LIN {X 0,Y 574.928,Z 413.278,A -85,B 0,C 180,E1 -2269.45,E2 -2269.45} C_VEL
LIN {X 0,Y 575.117,Z 397.956,A -85,B 0,C 180,E1 -2270.055,E2 -2270.055} C_VEL
LIN {X 0,Y 575.352,Z 381.203,A -85,B 0,C 180,E1 -2270.559,E2 -2270.559} C_VEL
LIN {X 0,Y 575.53,Z 364.973,A -85,B 0,C 180,E1 -2270.903,E2 -2270.903} C_VEL
LIN {X 0,Y 576.146,Z 164.419,A -85,B 0,C 180,E1 -2273.543,E2 -2273.543} C_VEL
LIN {X 0,Y 575.13,Z 158.184,A -85,B 0,C 180,E1 -2273.687,E2 -2273.687} C_VEL
LIN {X 0,Y 575.609,Z 123.808,A -85,B 0,C 180,E1 -2276.367,E2 -2276.367} C_VEL
LIN {X 0,Y 575.922,Z 94.132,A -85,B 0,C 180,E1 -2278.717,E2 -2278.717} C_VEL
LIN {X 0,Y 573.276,Z 85.388,A -85,B 0,C 180,E1 -2279.565,E2 -2279.565} C_VEL
LIN {X 0,Y 573.253,Z 85.395,A -85,B 0,C 180,E1 -2282.644,E2 -2282.644} C_VEL
LIN {X 0,Y 573.208,Z 85.394,A -85,B 0,C 180,E1 -2285.187,E2 -2285.187} C_VEL
LIN {X 0,Y 573.23,Z 85.39,A -85,B 0,C 180,E1 -2287.807,E2 -2287.807} C_VEL
LIN {X 0,Y 573.24,Z 85.397,A -85,B 0,C 180,E1 -2290.525,E2 -2290.525} C_VEL
LIN {X 0,Y 573.244,Z 85.387,A -85,B 0,C 180,E1 -2293.358,E2 -2293.358} C_VEL
LIN {X 0,Y 573.24,Z 85.396,A -85,B 0,C 180,E1 -2296.331,E2 -2296.331} C_VEL
LIN {X 0,Y 573.27,Z 85.383,A -85,B 0,C 180,E1 -2299.477,E2 -2299.477} C_VEL
LIN {X 0,Y 573.232,Z 85.396,A -85,B 0,C 180,E1 -2302.192,E2 -2302.192} C_VEL
LIN {X 0,Y 573.263,Z 85.385,A -85,B 0,C 180,E1 -2304.816,E2 -2304.816} C_VEL
LIN {X 0,Y 573.25,Z 85.385,A -85,B 0,C 180,E1 -2307.355,E2 -2307.355} C_VEL
LIN {X 0,Y 573.246,Z 85.39,A -85,B 0,C 180,E1 -2309.824,E2 -2309.824} C_VEL
LIN {X 0,Y 573.269,Z 85.391,A -85,B 0,C 180,E1 -2312.234,E2 -2312.234} C_VEL
LIN {X 0,Y 573.264,Z 85.383,A -85,B 0,C 180,E1 -2315.121,E2 -2315.121} C_VEL
LIN {X 0,Y 573.233,Z 85.392,A -85,B 0,C 180,E1 -2317.662,E2 -2317.662} C_VEL
LIN {X 0,Y 573.274,Z 85.383,A -85,B 0,C 180,E1 -2320.728,E2 -2320.728} C_VEL
LIN {X 0,Y 573.248,Z 85.391,A -85,B 0,C 180,E1 -2323.622,E2 -2323.622} C_VEL
LIN {X 0,Y 573.27,Z 85.392,A -85,B 0,C 180,E1 -2325.807,E2 -2325.807} C_VEL
LIN {X 0,Y 573.258,Z 85.384,A -85,B 0,C 180,E1 -2328.745,E2 -2328.745} C_VEL
LIN {X 0,Y 573.281,Z 85.387,A -85,B 0,C 180,E1 -2331.541,E2 -2331.541} C_VEL
LIN {X 0,Y 573.287,Z 85.382,A -85,B 0,C 180,E1 -2334.372,E2 -2334.372} C_VEL
LIN {X 0,Y 573.305,Z 85.385,A -85,B 0,C 180,E1 -2337.892,E2 -2337.892} C_VEL
LIN {X 0,Y 573.329,Z 85.375,A -85,B 0,C 180,E1 -2340.702,E2 -2340.702} C_VEL
LIN {X 0,Y 573.232,Z 85.397,A -85,B 0,C 180,E1 -2343.515,E2 -2343.515} C_VEL
LIN {X 0,Y 573.285,Z 85.389,A -85,B 0,C 180,E1 -2345.628,E2 -2345.628} C_VEL
LIN {X 0,Y 573.28,Z 85.381,A -85,B 0,C 180,E1 -2348.46,E2 -2348.46} C_VEL
LIN {X 0,Y 573.268,Z 85.391,A -85,B 0,C 180,E1 -2351.312,E2 -2351.312} C_VEL
LIN {X 0,Y 573.269,Z 85.383,A -85,B 0,C 180,E1 -2354.193,E2 -2354.193} C_VEL
LIN {X 0,Y 573.256,Z 85.391,A -85,B 0,C 180,E1 -2357.112,E2 -2357.112} C_VEL
LIN {X 0,Y 573.248,Z 85.386,A -85,B 0,C 180,E1 -2360.077,E2 -2360.077} C_VEL
LIN {X 0,Y 573.23,Z 85.396,A -85,B 0,C 180,E1 -2363.1,E2 -2363.1} C_VEL
LIN {X 0,Y 573.247,Z 85.386,A -85,B 0,C 180,E1 -2364.39,E2 -2364.39} C_VEL
LIN {X 0,Y 572.62,Z 85.471,A -85,B 0,C 180,E1 -2364.977,E2 -2364.977} C_VEL
LIN {X 0,Y 569.778,Z 85.828,A -85,B 0,C 180,E1 -2365.928,E2 -2365.928} C_VEL
LIN {X 0,Y 567.346,Z 86.132,A -85,B 0,C 180,E1 -2366.694,E2 -2366.694} C_VEL
LIN {X 0,Y 566.29,Z 86.26,A -85,B 0,C 180,E1 -2367.285,E2 -2367.285} C_VEL
LIN {X 0,Y 566.2,Z 86.268,A -85,B 0,C 180,E1 -2367.485,E2 -2367.485} C_VEL
LIN {X 0,Y 566.198,Z 86.265,A -85,B 0,C 180,E1 -2369.769,E2 -2369.769} C_VEL
LIN {X 0,Y 566.202,Z 86.265,A -85,B 0,C 180,E1 -2372.431,E2 -2372.431} C_VEL
LIN {X 0,Y 566.209,Z 86.272,A -85,B 0,C 180,E1 -2374.995,E2 -2374.995} C_VEL
LIN {X 0,Y 566.194,Z 86.267,A -85,B 0,C 180,E1 -2377.461,E2 -2377.461} C_VEL
LIN {X 0,Y 566.224,Z 86.261,A -85,B 0,C 180,E1 -2380.198,E2 -2380.198} C_VEL
LIN {X 0,Y 566.198,Z 86.271,A -85,B 0,C 180,E1 -2383.054,E2 -2383.054} C_VEL
LIN {X 0,Y 566.199,Z 86.264,A -85,B 0,C 180,E1 -2386.049,E2 -2386.049} C_VEL
LIN {X 0,Y 566.209,Z 86.271,A -85,B 0,C 180,E1 -2388.864,E2 -2388.864} C_VEL
LIN {X 0,Y 566.186,Z 86.265,A -85,B 0,C 180,E1 -2391.638,E2 -2391.638} C_VEL
LIN {X 0,Y 566.16,Z 86.272,A -85,B 0,C 180,E1 -2394.308,E2 -2394.308} C_VEL
LIN {X 0,Y 566.228,Z 86.266,A -85,B 0,C 180,E1 -2396.899,E2 -2396.899} C_VEL
LIN {X 0,Y 566.183,Z 86.266,A -85,B 0,C 180,E1 -2399.408,E2 -2399.408} C_VEL
LIN {X 0,Y 566.21,Z 86.263,A -85,B 0,C 180,E1 -2401.858,E2 -2401.858} C_VEL
LIN {X 0,Y 566.213,Z 86.268,A -85,B 0,C 180,E1 -2404.252,E2 -2404.252} C_VEL
LIN {X 0,Y 566.171,Z 86.273,A -85,B 0,C 180,E1 -2406.719,E2 -2406.719} C_VEL
LIN {X 0,Y 566.212,Z 86.263,A -85,B 0,C 180,E1 -2409.663,E2 -2409.663} C_VEL
LIN {X 0,Y 566.199,Z 86.269,A -85,B 0,C 180,E1 -2412.669,E2 -2412.669} C_VEL
LIN {X 0,Y 566.234,Z 86.26,A -85,B 0,C 180,E1 -2415.627,E2 -2415.627} C_VEL
LIN {X 0,Y 566.235,Z 86.263,A -85,B 0,C 180,E1 -2418.676,E2 -2418.676} C_VEL
LIN {X 0,Y 566.227,Z 86.261,A -85,B 0,C 180,E1 -2421.435,E2 -2421.435} C_VEL
LIN {X 0,Y 566.259,Z 86.264,A -85,B 0,C 180,E1 -2424.302,E2 -2424.302} C_VEL
LIN {X 0,Y 566.283,Z 86.259,A -85,B 0,C 180,E1 -2427.867,E2 -2427.867} C_VEL
LIN {X 0,Y 566.302,Z 86.252,A -85,B 0,C 180,E1 -2430.712,E2 -2430.712} C_VEL
LIN {X 0,Y 566.271,Z 86.255,A -85,B 0,C 180,E1 -2432.846,E2 -2432.846} C_VEL
LIN {X 0,Y 566.258,Z 86.262,A -85,B 0,C 180,E1 -2435.699,E2 -2435.699} C_VEL
LIN {X 0,Y 566.229,Z 86.261,A -85,B 0,C 180,E1 -2438.566,E2 -2438.566} C_VEL
LIN {X 0,Y 566.244,Z 86.262,A -85,B 0,C 180,E1 -2441.455,E2 -2441.455} C_VEL
LIN {X 0,Y 566.236,Z 86.26,A -85,B 0,C 180,E1 -2444.507,E2 -2444.507} C_VEL
LIN {X 0,Y 566.201,Z 86.267,A -85,B 0,C 180,E1 -2447.332,E2 -2447.332} C_VEL
LIN {X 0,Y 566.214,Z 86.263,A -85,B 0,C 180,E1 -2450.338,E2 -2450.338} C_VEL
LIN {X 0,Y 566.175,Z 86.271,A -85,B 0,C 180,E1 -2453.282,E2 -2453.282} C_VEL
LIN {X 0,Y 566.217,Z 86.269,A -85,B 0,C 180,E1 -2455.749,E2 -2455.749} C_VEL
LIN {X 0,Y 566.205,Z 86.264,A -85,B 0,C 180,E1 -2458.202,E2 -2458.202} C_VEL
LIN {X 0,Y 566.192,Z 86.268,A -85,B 0,C 180,E1 -2461.077,E2 -2461.077} C_VEL
LIN {X 0,Y 566.214,Z 86.267,A -85,B 0,C 180,E1 -2463.734,E2 -2463.734} C_VEL
LIN {X 0,Y 566.201,Z 86.264,A -85,B 0,C 180,E1 -2466.57,E2 -2466.57} C_VEL
LIN {X 0,Y 566.216,Z 86.266,A -85,B 0,C 180,E1 -2469.686,E2 -2469.686} C_VEL
LIN {X 0,Y 566.205,Z 86.267,A -85,B 0,C 180,E1 -2472.918,E2 -2472.918} C_VEL
LIN {X 0,Y 566.197,Z 86.264,A -85,B 0,C 180,E1 -2476.049,E2 -2476.049} C_VEL
LIN {X 0,Y 566.206,Z 86.273,A -85,B 0,C 180,E1 -2479.215,E2 -2479.215} C_VEL
LIN {X 0,Y 566.189,Z 86.268,A -85,B 0,C 180,E1 -2481.637,E2 -2481.637} C_VEL
LIN {X 0,Y 566.195,Z 86.265,A -85,B 0,C 180,E1 -2484.31,E2 -2484.31} C_VEL
LIN {X 0,Y 566.223,Z 86.268,A -85,B 0,C 180,E1 -2486.898,E2 -2486.898} C_VEL
LIN {X 0,Y 566.184,Z 86.271,A -85,B 0,C 180,E1 -2489.407,E2 -2489.407} C_VEL
LIN {X 0,Y 566.216,Z 86.264,A -85,B 0,C 180,E1 -2491.858,E2 -2491.858} C_VEL
LIN {X 0,Y 566.213,Z 86.266,A -85,B 0,C 180,E1 -2494.251,E2 -2494.251} C_VEL
LIN {X 0,Y 566.197,Z 86.269,A -85,B 0,C 180,E1 -2496.075,E2 -2496.075} C_VEL
LIN {X 0,Y 567.227,Z 89.177,A -85,B 0,C 180,E1 -2496.169,E2 -2496.169} C_VEL
LIN {X 0,Y 569.661,Z 94.835,A -85,B 0,C 180,E1 -2496.361,E2 -2496.361} C_VEL
LIN {X 0,Y 568.867,Z 283.383,A -85,B 0,C 180,E1 -2498.863,E2 -2498.863} C_VEL
LIN {X 0,Y 568.754,Z 299.599,A -85,B 0,C 180,E1 -2499.191,E2 -2499.191} C_VEL
LIN {X 0,Y 568.499,Z 315.266,A -85,B 0,C 180,E1 -2499.654,E2 -2499.654} C_VEL
LIN {X 0,Y 568.295,Z 327.963,A -85,B 0,C 180,E1 -2500.132,E2 -2500.132} C_VEL
LIN {X 0,Y 567.998,Z 341.858,A -85,B 0,C 180,E1 -2500.765,E2 -2500.765} C_VEL
LIN {X 0,Y 567.689,Z 356.768,A -85,B 0,C 180,E1 -2501.597,E2 -2501.597} C_VEL
LIN {X 0,Y 567.395,Z 369.444,A -85,B 0,C 180,E1 -2502.444,E2 -2502.444} C_VEL
LIN {X 0,Y 567.154,Z 381.162,A -85,B 0,C 180,E1 -2503.348,E2 -2503.348} C_VEL
LIN {X 0,Y 566.863,Z 392.522,A -85,B 0,C 180,E1 -2504.356,E2 -2504.356} C_VEL
LIN {X 0,Y 566.634,Z 404.905,A -85,B 0,C 180,E1 -2505.637,E2 -2505.637} C_VEL
LIN {X 0,Y 566.379,Z 415.329,A -85,B 0,C 180,E1 -2506.911,E2 -2506.911} C_VEL
LIN {X 0,Y 566.221,Z 424.31,A -85,B 0,C 180,E1 -2508.182,E2 -2508.182} C_VEL
LIN {X 0,Y 566.118,Z 432.007,A -85,B 0,C 180,E1 -2509.449,E2 -2509.449} C_VEL
LIN {X 0,Y 566.005,Z 438.589,A -85,B 0,C 180,E1 -2510.711,E2 -2510.711} C_VEL
LIN {X 0,Y 565.979,Z 444.894,A -85,B 0,C 180,E1 -2512.149,E2 -2512.149} C_VEL
LIN {X 0,Y 565.92,Z 449.999,A -85,B 0,C 180,E1 -2513.583,E2 -2513.583} C_VEL
LIN {X 0,Y 565.86,Z 453.972,A -85,B 0,C 180,E1 -2515.012,E2 -2515.012} C_VEL
LIN {X 0,Y 565.911,Z 456.887,A -85,B 0,C 180,E1 -2516.44,E2 -2516.44} C_VEL
LIN {X 0,Y 565.829,Z 458.84,A -85,B 0,C 180,E1 -2517.864,E2 -2517.864} C_VEL
LIN {X 0,Y 565.839,Z 459.811,A -85,B 0,C 180,E1 -2519.288,E2 -2519.288} C_VEL
LIN {X 0,Y 565.841,Z 459.839,A -85,B 0,C 180,E1 -2520.712,E2 -2520.712} C_VEL
LIN {X 0,Y 565.829,Z 458.925,A -85,B 0,C 180,E1 -2522.135,E2 -2522.135} C_VEL
LIN {X 0,Y 565.91,Z 457.029,A -85,B 0,C 180,E1 -2523.56,E2 -2523.56} C_VEL
LIN {X 0,Y 565.858,Z 454.187,A -85,B 0,C 180,E1 -2524.988,E2 -2524.988} C_VEL
LIN {X 0,Y 565.948,Z 449.836,A -85,B 0,C 180,E1 -2526.56,E2 -2526.56} C_VEL
LIN {X 0,Y 565.99,Z 443.787,A -85,B 0,C 180,E1 -2528.21,E2 -2528.21} C_VEL
LIN {X 0,Y 566.034,Z 437.256,A -85,B 0,C 180,E1 -2529.649,E2 -2529.649} C_VEL
LIN {X 0,Y 566.18,Z 429.121,A -85,B 0,C 180,E1 -2531.147,E2 -2531.147} C_VEL
LIN {X 0,Y 566.322,Z 420.049,A -85,B 0,C 180,E1 -2532.543,E2 -2532.543} C_VEL
LIN {X 0,Y 566.514,Z 410.291,A -85,B 0,C 180,E1 -2533.816,E2 -2533.816} C_VEL
LIN {X 0,Y 566.701,Z 400.453,A -85,B 0,C 180,E1 -2534.932,E2 -2534.932} C_VEL
LIN {X 0,Y 566.901,Z 391.505,A -85,B 0,C 180,E1 -2535.827,E2 -2535.827} C_VEL
LIN {X 0,Y 567.147,Z 380.013,A -85,B 0,C 180,E1 -2536.837,E2 -2536.837} C_VEL
LIN {X 0,Y 567.449,Z 367.853,A -85,B 0,C 180,E1 -2537.761,E2 -2537.761} C_VEL
LIN {X 0,Y 567.762,Z 353.698,A -85,B 0,C 180,E1 -2538.68,E2 -2538.68} C_VEL
LIN {X 0,Y 568.039,Z 339.87,A -85,B 0,C 180,E1 -2539.421,E2 -2539.421} C_VEL
LIN {X 0,Y 568.304,Z 326.571,A -85,B 0,C 180,E1 -2540.017,E2 -2540.017} C_VEL
LIN {X 0,Y 568.611,Z 310.214,A -85,B 0,C 180,E1 -2540.602,E2 -2540.602} C_VEL
LIN {X 0,Y 568.775,Z 295.187,A -85,B 0,C 180,E1 -2540.998,E2 -2540.998} C_VEL
LIN {X 0,Y 568.884,Z 281.636,A -85,B 0,C 180,E1 -2541.254,E2 -2541.254} C_VEL
LIN {X 0,Y 569.594,Z 95.156,A -85,B 0,C 180,E1 -2543.726,E2 -2543.726} C_VEL
LIN {X 0,Y 569.036,Z 93.275,A -85,B 0,C 180,E1 -2543.778,E2 -2543.778} C_VEL
LIN {X 0,Y 566.316,Z 87.098,A -85,B 0,C 180,E1 -2543.991,E2 -2543.991} C_VEL
LIN {X 0,Y 566.14,Z 86.277,A -85,B 0,C 180,E1 -2544.028,E2 -2544.028} C_VEL
LIN {X 0,Y 566.169,Z 86.275,A -85,B 0,C 180,E1 -2546.65,E2 -2546.65} C_VEL
LIN {X 0,Y 566.158,Z 86.272,A -85,B 0,C 180,E1 -2549.771,E2 -2549.771} C_VEL
LIN {X 0,Y 566.194,Z 86.272,A -85,B 0,C 180,E1 -2552.428,E2 -2552.428} C_VEL
LIN {X 0,Y 566.178,Z 86.272,A -85,B 0,C 180,E1 -2554.989,E2 -2554.989} C_VEL
LIN {X 0,Y 566.192,Z 86.267,A -85,B 0,C 180,E1 -2557.461,E2 -2557.461} C_VEL
LIN {X 0,Y 566.207,Z 86.271,A -85,B 0,C 180,E1 -2560.199,E2 -2560.199} C_VEL
LIN {X 0,Y 566.198,Z 86.266,A -85,B 0,C 180,E1 -2563.054,E2 -2563.054} C_VEL
LIN {X 0,Y 566.2,Z 86.273,A -85,B 0,C 180,E1 -2566.048,E2 -2566.048} C_VEL
LIN {X 0,Y 566.205,Z 86.266,A -85,B 0,C 180,E1 -2569.214,E2 -2569.214} C_VEL
LIN {X 0,Y 566.188,Z 86.274,A -85,B 0,C 180,E1 -2571.636,E2 -2571.636} C_VEL
LIN {X 0,Y 566.164,Z 86.273,A -85,B 0,C 180,E1 -2574.308,E2 -2574.308} C_VEL
LIN {X 0,Y 566.23,Z 86.267,A -85,B 0,C 180,E1 -2576.898,E2 -2576.898} C_VEL
LIN {X 0,Y 566.182,Z 86.279,A -85,B 0,C 180,E1 -2579.407,E2 -2579.407} C_VEL
LIN {X 0,Y 566.226,Z 86.394,A -85,B 0,C 180,E1 -2580.324,E2 -2580.324} C_VEL
LIN {X 0,Y 569.015,Z 96.641,A -85,B 0,C 180,E1 -2581.274,E2 -2581.274} C_VEL
LIN {X 0,Y 568.654,Z 132.486,A -85,B 0,C 180,E1 -2584.074,E2 -2584.074} C_VEL
LIN {X 0,Y 568.402,Z 157.927,A -85,B 0,C 180,E1 -2586.031,E2 -2586.031} C_VEL
LIN {X 0,Y 569.69,Z 167.303,A -85,B 0,C 180,E1 -2586.217,E2 -2586.217} C_VEL
LIN {X 0,Y 568.884,Z 364.907,A -85,B 0,C 180,E1 -2588.84,E2 -2588.84} C_VEL
LIN {X 0,Y 568.702,Z 381.158,A -85,B 0,C 180,E1 -2589.188,E2 -2589.188} C_VEL
LIN {X 0,Y 568.44,Z 397.926,A -85,B 0,C 180,E1 -2589.698,E2 -2589.698} C_VEL
LIN {X 0,Y 568.206,Z 413.659,A -85,B 0,C 180,E1 -2590.329,E2 -2590.329} C_VEL
LIN {X 0,Y 567.901,Z 428.026,A -85,B 0,C 180,E1 -2591.043,E2 -2591.043} C_VEL
LIN {X 0,Y 567.532,Z 443.265,A -85,B 0,C 180,E1 -2591.965,E2 -2591.965} C_VEL
LIN {X 0,Y 567.19,Z 457.209,A -85,B 0,C 180,E1 -2592.978,E2 -2592.978} C_VEL
LIN {X 0,Y 566.916,Z 471.063,A -85,B 0,C 180,E1 -2594.173,E2 -2594.173} C_VEL
LIN {X 0,Y 566.632,Z 482.615,A -85,B 0,C 180,E1 -2595.339,E2 -2595.339} C_VEL
LIN {X 0,Y 566.435,Z 494.334,A -85,B 0,C 180,E1 -2596.73,E2 -2596.73} C_VEL
LIN {X 0,Y 566.239,Z 504.668,A -85,B 0,C 180,E1 -2598.182,E2 -2598.182} C_VEL
LIN {X 0,Y 566.124,Z 513.281,A -85,B 0,C 180,E1 -2599.629,E2 -2599.629} C_VEL
LIN {X 0,Y 566.002,Z 520.488,A -85,B 0,C 180,E1 -2601.07,E2 -2601.07} C_VEL
LIN {X 0,Y 565.967,Z 526.464,A -85,B 0,C 180,E1 -2602.508,E2 -2602.508} C_VEL
LIN {X 0,Y 565.916,Z 531.186,A -85,B 0,C 180,E1 -2603.94,E2 -2603.94} C_VEL
LIN {X 0,Y 565.91,Z 535.635,A -85,B 0,C 180,E1 -2605.726,E2 -2605.726} C_VEL
LIN {X 0,Y 565.867,Z 538.089,A -85,B 0,C 180,E1 -2607.152,E2 -2607.152} C_VEL
LIN {X 0,Y 565.843,Z 539.479,A -85,B 0,C 180,E1 -2608.576,E2 -2608.576} C_VEL
LIN {X 0,Y 565.834,Z 540,A -85,B 0,C 180,E1 -2610,E2 -2610} C_VEL
LIN {X 0,Y 565.843,Z 539.48,A -85,B 0,C 180,E1 -2611.423,E2 -2611.423} C_VEL
LIN {X 0,Y 565.867,Z 538.089,A -85,B 0,C 180,E1 -2612.847,E2 -2612.847} C_VEL
LIN {X 0,Y 565.91,Z 535.637,A -85,B 0,C 180,E1 -2614.273,E2 -2614.273} C_VEL
LIN {X 0,Y 565.915,Z 531.19,A -85,B 0,C 180,E1 -2616.059,E2 -2616.059} C_VEL
LIN {X 0,Y 565.969,Z 526.47,A -85,B 0,C 180,E1 -2617.491,E2 -2617.491} C_VEL
LIN {X 0,Y 566.011,Z 520.492,A -85,B 0,C 180,E1 -2618.928,E2 -2618.928} C_VEL
LIN {X 0,Y 566.123,Z 513.286,A -85,B 0,C 180,E1 -2620.37,E2 -2620.37} C_VEL
LIN {X 0,Y 566.237,Z 504.676,A -85,B 0,C 180,E1 -2621.817,E2 -2621.817} C_VEL
LIN {X 0,Y 566.434,Z 494.342,A -85,B 0,C 180,E1 -2623.269,E2 -2623.269} C_VEL
LIN {X 0,Y 566.617,Z 482.669,A -85,B 0,C 180,E1 -2624.655,E2 -2624.655} C_VEL
LIN {X 0,Y 566.914,Z 471.072,A -85,B 0,C 180,E1 -2625.826,E2 -2625.826} C_VEL
LIN {X 0,Y 567.223,Z 457.222,A -85,B 0,C 180,E1 -2627.02,E2 -2627.02} C_VEL
LIN {X 0,Y 567.581,Z 443.28,A -85,B 0,C 180,E1 -2628.032,E2 -2628.032} C_VEL
LIN {X 0,Y 567.877,Z 429.716,A -85,B 0,C 180,E1 -2628.863,E2 -2628.863} C_VEL
LIN {X 0,Y 568.154,Z 415.368,A -85,B 0,C 180,E1 -2629.592,E2 -2629.592} C_VEL
LIN {X 0,Y 568.42,Z 399.254,A -85,B 0,C 180,E1 -2630.254,E2 -2630.254} C_VEL
LIN {X 0,Y 568.726,Z 383.034,A -85,B 0,C 180,E1 -2630.762,E2 -2630.762} C_VEL
LIN {X 0,Y 568.892,Z 366.461,A -85,B 0,C 180,E1 -2631.135,E2 -2631.135} C_VEL
LIN {X 0,Y 569.65,Z 175.195,A -85,B 0,C 180,E1 -2633.678,E2 -2633.678} C_VEL
LIN {X 0,Y 569.486,Z 164.584,A -85,B 0,C 180,E1 -2633.827,E2 -2633.827} C_VEL
LIN {X 0,Y 568.424,Z 158.163,A -85,B 0,C 180,E1 -2633.969,E2 -2633.969} C_VEL
LIN {X 0,Y 568.936,Z 123.563,A -85,B 0,C 180,E1 -2636.689,E2 -2636.689} C_VEL
LIN {X 0,Y 569.296,Z 96.342,A -85,B 0,C 180,E1 -2638.871,E2 -2638.871} C_VEL
LIN {X 0,Y 566.225,Z 86.267,A -85,B 0,C 180,E1 -2639.869,E2 -2639.869} C_VEL
LIN {X 0,Y 566.226,Z 86.266,A -85,B 0,C 180,E1 -2643.101,E2 -2643.101} C_VEL
LIN {X 0,Y 566.161,Z 86.27,A -85,B 0,C 180,E1 -2645.692,E2 -2645.692} C_VEL
LIN {X 0,Y 566.207,Z 86.273,A -85,B 0,C 180,E1 -2648.558,E2 -2648.558} C_VEL
LIN {X 0,Y 566.179,Z 86.268,A -85,B 0,C 180,E1 -2651.138,E2 -2651.138} C_VEL
LIN {X 0,Y 566.196,Z 86.268,A -85,B 0,C 180,E1 -2654.035,E2 -2654.035} C_VEL
LIN {X 0,Y 566.197,Z 86.265,A -85,B 0,C 180,E1 -2657.083,E2 -2657.083} C_VEL
LIN {X 0,Y 566.223,Z 86.263,A -85,B 0,C 180,E1 -2659.802,E2 -2659.802} C_VEL
LIN {X 0,Y 566.194,Z 86.269,A -85,B 0,C 180,E1 -2662.599,E2 -2662.599} C_VEL
LIN {X 0,Y 566.216,Z 86.261,A -85,B 0,C 180,E1 -2665.183,E2 -2665.183} C_VEL
LIN {X 0,Y 566.228,Z 86.263,A -85,B 0,C 180,E1 -2667.743,E2 -2667.743} C_VEL
LIN {X 0,Y 566.2,Z 86.27,A -85,B 0,C 180,E1 -2670.328,E2 -2670.328} C_VEL
LIN {X 0,Y 566.207,Z 86.263,A -85,B 0,C 180,E1 -2673.34,E2 -2673.34} C_VEL
LIN {X 0,Y 566.195,Z 86.27,A -85,B 0,C 180,E1 -2675.819,E2 -2675.819} C_VEL
LIN {X 0,Y 566.204,Z 86.263,A -85,B 0,C 180,E1 -2678.902,E2 -2678.902} C_VEL
LIN {X 0,Y 566.204,Z 86.263,A -85,B 0,C 180,E1 -2681.172,E2 -2681.172} C_VEL
LIN {X 0,Y 566.212,Z 86.264,A -85,B 0,C 180,E1 -2683.412,E2 -2683.412} C_VEL
LIN {X 0,Y 566.196,Z 86.267,A -85,B 0,C 180,E1 -2686.359,E2 -2686.359} C_VEL
LIN {X 0,Y 566.23,Z 86.26,A -85,B 0,C 180,E1 -2688.675,E2 -2688.675} C_VEL
LIN {X 0,Y 566.224,Z 86.265,A -85,B 0,C 180,E1 -2691.434,E2 -2691.434} C_VEL
LIN {X 0,Y 566.255,Z 86.258,A -85,B 0,C 180,E1 -2694.302,E2 -2694.302} C_VEL
LIN {X 0,Y 566.276,Z 86.261,A -85,B 0,C 180,E1 -2697.866,E2 -2697.866} C_VEL
LIN {X 0,Y 566.299,Z 86.251,A -85,B 0,C 180,E1 -2700.711,E2 -2700.711} C_VEL
LIN {X 0,Y 566.27,Z 86.255,A -85,B 0,C 180,E1 -2702.846,E2 -2702.846} C_VEL
LIN {X 0,Y 566.253,Z 86.264,A -85,B 0,C 180,E1 -2705.698,E2 -2705.698} C_VEL
LIN {X 0,Y 566.224,Z 86.261,A -85,B 0,C 180,E1 -2708.566,E2 -2708.566} C_VEL
LIN {X 0,Y 566.238,Z 86.269,A -85,B 0,C 180,E1 -2711.454,E2 -2711.454} C_VEL
LIN {X 0,Y 566.23,Z 86.26,A -85,B 0,C 180,E1 -2714.507,E2 -2714.507} C_VEL
LIN {X 0,Y 566.2,Z 86.274,A -85,B 0,C 180,E1 -2717.332,E2 -2717.332} C_VEL
LIN {X 0,Y 566.21,Z 86.262,A -85,B 0,C 180,E1 -2720.337,E2 -2720.337} C_VEL
LIN {X 0,Y 566.186,Z 86.272,A -85,B 0,C 180,E1 -2723.404,E2 -2723.404} C_VEL
LIN {X 0,Y 566.21,Z 86.264,A -85,B 0,C 180,E1 -2725.749,E2 -2725.749} C_VEL
LIN {X 0,Y 566.2,Z 86.268,A -85,B 0,C 180,E1 -2727.485,E2 -2727.485} C_VEL
LIN {X 0,Y 565.519,Z 86.351,A -85,B 0,C 180,E1 -2728.079,E2 -2728.079} C_VEL
LIN {X 0,Y 562.654,Z 86.714,A -85,B 0,C 180,E1 -2729.042,E2 -2729.042} C_VEL
LIN {X 0,Y 560.246,Z 87.009,A -85,B 0,C 180,E1 -2729.818,E2 -2729.818} C_VEL
LIN {X 0,Y 559.221,Z 87.134,A -85,B 0,C 180,E1 -2730.417,E2 -2730.417} C_VEL
LIN {X 0,Y 559.142,Z 87.146,A -85,B 0,C 180,E1 -2730.619,E2 -2730.619} C_VEL
LIN {X 0,Y 559.161,Z 87.143,A -85,B 0,C 180,E1 -2733.575,E2 -2733.575} C_VEL
LIN {X 0,Y 559.166,Z 87.142,A -85,B 0,C 180,E1 -2736.449,E2 -2736.449} C_VEL
LIN {X 0,Y 559.176,Z 87.148,A -85,B 0,C 180,E1 -2738.934,E2 -2738.934} C_VEL
LIN {X 0,Y 559.188,Z 87.137,A -85,B 0,C 180,E1 -2741.768,E2 -2741.768} C_VEL
LIN {X 0,Y 559.136,Z 87.152,A -85,B 0,C 180,E1 -2744.74,E2 -2744.74} C_VEL
LIN {X 0,Y 559.162,Z 87.143,A -85,B 0,C 180,E1 -2747.257,E2 -2747.257} C_VEL
LIN {X 0,Y 559.182,Z 87.139,A -85,B 0,C 180,E1 -2750.135,E2 -2750.135} C_VEL
LIN {X 0,Y 559.138,Z 87.15,A -85,B 0,C 180,E1 -2752.892,E2 -2752.892} C_VEL
LIN {X 0,Y 559.164,Z 87.142,A -85,B 0,C 180,E1 -2756.051,E2 -2756.051} C_VEL
LIN {X 0,Y 559.159,Z 87.144,A -85,B 0,C 180,E1 -2758.982,E2 -2758.982} C_VEL
LIN {X 0,Y 559.166,Z 87.14,A -85,B 0,C 180,E1 -2761.619,E2 -2761.619} C_VEL
LIN {X 0,Y 559.18,Z 87.14,A -85,B 0,C 180,E1 -2763.903,E2 -2763.903} C_VEL
LIN {X 0,Y 559.15,Z 87.15,A -85,B 0,C 180,E1 -2766.569,E2 -2766.569} C_VEL
LIN {X 0,Y 559.179,Z 87.138,A -85,B 0,C 180,E1 -2769.396,E2 -2769.396} C_VEL
LIN {X 0,Y 559.145,Z 87.143,A -85,B 0,C 180,E1 -2771.686,E2 -2771.686} C_VEL
LIN {X 0,Y 559.165,Z 87.144,A -85,B 0,C 180,E1 -2773.948,E2 -2773.948} C_VEL
LIN {X 0,Y 559.171,Z 87.147,A -85,B 0,C 180,E1 -2776.185,E2 -2776.185} C_VEL
LIN {X 0,Y 559.195,Z 87.136,A -85,B 0,C 180,E1 -2779.134,E2 -2779.134} C_VEL
LIN {X 0,Y 559.204,Z 87.142,A -85,B 0,C 180,E1 -2782.054,E2 -2782.054} C_VEL
LIN {X 0,Y 559.251,Z 87.129,A -85,B 0,C 180,E1 -2784.954,E2 -2784.954} C_VEL
LIN {X 0,Y 559.254,Z 87.134,A -85,B 0,C 180,E1 -2787.84,E2 -2787.84} C_VEL
LIN {X 0,Y 559.273,Z 87.128,A -85,B 0,C 180,E1 -2790.72,E2 -2790.72} C_VEL
LIN {X 0,Y 559.238,Z 87.131,A -85,B 0,C 180,E1 -2792.882,E2 -2792.882} C_VEL
LIN {X 0,Y 559.228,Z 87.139,A -85,B 0,C 180,E1 -2795.771,E2 -2795.771} C_VEL
LIN {X 0,Y 559.187,Z 87.138,A -85,B 0,C 180,E1 -2798.675,E2 -2798.675} C_VEL
LIN {X 0,Y 559.207,Z 87.14,A -85,B 0,C 180,E1 -2801.601,E2 -2801.601} C_VEL
LIN {X 0,Y 559.202,Z 87.136,A -85,B 0,C 180,E1 -2804.596,E2 -2804.596} C_VEL
LIN {X 0,Y 559.161,Z 87.147,A -85,B 0,C 180,E1 -2807.557,E2 -2807.557} C_VEL
LIN {X 0,Y 559.174,Z 87.147,A -85,B 0,C 180,E1 -2809.838,E2 -2809.838} C_VEL
LIN {X 0,Y 559.143,Z 87.145,A -85,B 0,C 180,E1 -2812.153,E2 -2812.153} C_VEL
LIN {X 0,Y 559.179,Z 87.143,A -85,B 0,C 180,E1 -2815.298,E2 -2815.298} C_VEL
LIN {X 0,Y 559.182,Z 87.145,A -85,B 0,C 180,E1 -2817.713,E2 -2817.713} C_VEL
LIN {X 0,Y 559.155,Z 87.142,A -85,B 0,C 180,E1 -2820.183,E2 -2820.183} C_VEL
LIN {X 0,Y 559.178,Z 87.139,A -85,B 0,C 180,E1 -2822.714,E2 -2822.714} C_VEL
LIN {X 0,Y 559.13,Z 87.152,A -85,B 0,C 180,E1 -2825.324,E2 -2825.324} C_VEL
LIN {X 0,Y 559.133,Z 87.145,A -85,B 0,C 180,E1 -2828.018,E2 -2828.018} C_VEL
LIN {X 0,Y 559.158,Z 87.143,A -85,B 0,C 180,E1 -2830.813,E2 -2830.813} C_VEL
LIN {X 0,Y 559.144,Z 87.146,A -85,B 0,C 180,E1 -2833.734,E2 -2833.734} C_VEL
LIN {X 0,Y 559.147,Z 87.145,A -85,B 0,C 180,E1 -2836.804,E2 -2836.804} C_VEL
LIN {X 0,Y 559.158,Z 87.151,A -85,B 0,C 180,E1 -2839.188,E2 -2839.188} C_VEL
LIN {X 0,Y 559.136,Z 87.144,A -85,B 0,C 180,E1 -2841.983,E2 -2841.983} C_VEL
LIN {X 0,Y 559.149,Z 87.148,A -85,B 0,C 180,E1 -2844.785,E2 -2844.785} C_VEL
LIN {X 0,Y 559.159,Z 87.147,A -85,B 0,C 180,E1 -2847.365,E2 -2847.365} C_VEL
LIN {X 0,Y 559.152,Z 87.143,A -85,B 0,C 180,E1 -2850.143,E2 -2850.143} C_VEL
LIN {X 0,Y 559.173,Z 87.148,A -85,B 0,C 180,E1 -2853.098,E2 -2853.098} C_VEL
LIN {X 0,Y 559.18,Z 87.144,A -85,B 0,C 180,E1 -2855.765,E2 -2855.765} C_VEL
LIN {X 0,Y 560.191,Z 90.027,A -85,B 0,C 180,E1 -2855.861,E2 -2855.861} C_VEL
LIN {X 0,Y 563.093,Z 96.361,A -85,B 0,C 180,E1 -2856.089,E2 -2856.089} C_VEL
LIN {X 0,Y 562.35,Z 268.953,A -85,B 0,C 180,E1 -2858.414,E2 -2858.414} C_VEL
LIN {X 0,Y 562.17,Z 290.5,A -85,B 0,C 180,E1 -2858.743,E2 -2858.743} C_VEL
LIN {X 0,Y 561.965,Z 305.908,A -85,B 0,C 180,E1 -2859.119,E2 -2859.119} C_VEL
LIN {X 0,Y 561.715,Z 321.235,A -85,B 0,C 180,E1 -2859.618,E2 -2859.618} C_VEL
LIN {X 0,Y 561.416,Z 336.076,A -85,B 0,C 180,E1 -2860.245,E2 -2860.245} C_VEL
LIN {X 0,Y 561.115,Z 348.788,A -85,B 0,C 180,E1 -2860.9,E2 -2860.9} C_VEL
LIN {X 0,Y 560.755,Z 362.596,A -85,B 0,C 180,E1 -2861.74,E2 -2861.74} C_VEL
LIN {X 0,Y 560.353,Z 377.788,A -85,B 0,C 180,E1 -2862.858,E2 -2862.858} C_VEL
LIN {X 0,Y 559.998,Z 388.564,A -85,B 0,C 180,E1 -2863.785,E2 -2863.785} C_VEL
LIN {X 0,Y 559.834,Z 398.042,A -85,B 0,C 180,E1 -2864.715,E2 -2864.715} C_VEL
LIN {X 0,Y 559.583,Z 407.996,A -85,B 0,C 180,E1 -2865.824,E2 -2865.824} C_VEL
LIN {X 0,Y 559.341,Z 416.68,A -85,B 0,C 180,E1 -2866.929,E2 -2866.929} C_VEL
LIN {X 0,Y 559.191,Z 425.49,A -85,B 0,C 180,E1 -2868.215,E2 -2868.215} C_VEL
LIN {X 0,Y 559.067,Z 433.035,A -85,B 0,C 180,E1 -2869.497,E2 -2869.497} C_VEL
LIN {X 0,Y 558.941,Z 440.32,A -85,B 0,C 180,E1 -2870.957,E2 -2870.957} C_VEL
LIN {X 0,Y 558.899,Z 446.276,A -85,B 0,C 180,E1 -2872.413,E2 -2872.413} C_VEL
LIN {X 0,Y 558.821,Z 450.583,A -85,B 0,C 180,E1 -2873.699,E2 -2873.699} C_VEL
LIN {X 0,Y 558.777,Z 453.977,A -85,B 0,C 180,E1 -2874.949,E2 -2874.949} C_VEL
LIN {X 0,Y 558.82,Z 456.884,A -85,B 0,C 180,E1 -2876.395,E2 -2876.395} C_VEL
LIN {X 0,Y 558.736,Z 458.832,A -85,B 0,C 180,E1 -2877.837,E2 -2877.837} C_VEL
LIN {X 0,Y 558.74,Z 459.805,A -85,B 0,C 180,E1 -2879.279,E2 -2879.279} C_VEL
LIN {X 0,Y 558.741,Z 459.833,A -85,B 0,C 180,E1 -2880.721,E2 -2880.721} C_VEL
LIN {X 0,Y 558.736,Z 458.917,A -85,B 0,C 180,E1 -2882.162,E2 -2882.162} C_VEL
LIN {X 0,Y 558.819,Z 457.024,A -85,B 0,C 180,E1 -2883.605,E2 -2883.605} C_VEL
LIN {X 0,Y 558.774,Z 454.178,A -85,B 0,C 180,E1 -2885.051,E2 -2885.051} C_VEL
LIN {X 0,Y 558.884,Z 449.095,A -85,B 0,C 180,E1 -2886.861,E2 -2886.861} C_VEL
LIN {X 0,Y 558.914,Z 443.776,A -85,B 0,C 180,E1 -2888.314,E2 -2888.314} C_VEL
LIN {X 0,Y 558.971,Z 437.246,A -85,B 0,C 180,E1 -2889.772,E2 -2889.772} C_VEL
LIN {X 0,Y 559.144,Z 428.701,A -85,B 0,C 180,E1 -2891.361,E2 -2891.361} C_VEL
LIN {X 0,Y 559.32,Z 418.689,A -85,B 0,C 180,E1 -2892.887,E2 -2892.887} C_VEL
LIN {X 0,Y 559.522,Z 410.275,A -85,B 0,C 180,E1 -2893.992,E2 -2893.992} C_VEL
LIN {X 0,Y 559.75,Z 400.624,A -85,B 0,C 180,E1 -2895.102,E2 -2895.102} C_VEL
LIN {X 0,Y 559.97,Z 391.488,A -85,B 0,C 180,E1 -2896.028,E2 -2896.028} C_VEL
LIN {X 0,Y 560.238,Z 381.107,A -85,B 0,C 180,E1 -2896.957,E2 -2896.957} C_VEL
LIN {X 0,Y 560.533,Z 371.13,A -85,B 0,C 180,E1 -2897.743,E2 -2897.743} C_VEL
LIN {X 0,Y 560.818,Z 359.609,A -85,B 0,C 180,E1 -2898.541,E2 -2898.541} C_VEL
LIN {X 0,Y 561.169,Z 345.4,A -85,B 0,C 180,E1 -2899.383,E2 -2899.383} C_VEL
LIN {X 0,Y 561.522,Z 330.8,A -85,B 0,C 180,E1 -2900.08,E2 -2900.08} C_VEL
LIN {X 0,Y 561.771,Z 317.424,A -85,B 0,C 180,E1 -2900.601,E2 -2900.601} C_VEL
LIN {X 0,Y 562.035,Z 302.156,A -85,B 0,C 180,E1 -2901.07,E2 -2901.07} C_VEL
LIN {X 0,Y 562.155,Z 285.465,A -85,B 0,C 180,E1 -2901.425,E2 -2901.425} C_VEL
LIN {X 0,Y 563.093,Z 97.418,A -85,B 0,C 180,E1 -2903.985,E2 -2903.985} C_VEL
LIN {X 0,Y 562.696,Z 95.555,A -85,B 0,C 180,E1 -2904.031,E2 -2904.031} C_VEL
LIN {X 0,Y 559.278,Z 88.023,A -85,B 0,C 180,E1 -2904.3,E2 -2904.3} C_VEL
LIN {X 0,Y 559.095,Z 87.155,A -85,B 0,C 180,E1 -2904.339,E2 -2904.339} C_VEL
LIN {X 0,Y 559.113,Z 87.156,A -85,B 0,C 180,E1 -2906.905,E2 -2906.905} C_VEL
LIN {X 0,Y 559.109,Z 87.15,A -85,B 0,C 180,E1 -2909.849,E2 -2909.849} C_VEL
LIN {X 0,Y 559.149,Z 87.152,A -85,B 0,C 180,E1 -2912.716,E2 -2912.716} C_VEL
LIN {X 0,Y 559.124,Z 87.148,A -85,B 0,C 180,E1 -2915.324,E2 -2915.324} C_VEL
LIN {X 0,Y 559.129,Z 87.15,A -85,B 0,C 180,E1 -2918.018,E2 -2918.018} C_VEL
LIN {X 0,Y 559.156,Z 87.145,A -85,B 0,C 180,E1 -2920.812,E2 -2920.812} C_VEL
LIN {X 0,Y 559.139,Z 87.148,A -85,B 0,C 180,E1 -2923.734,E2 -2923.734} C_VEL
LIN {X 0,Y 559.15,Z 87.144,A -85,B 0,C 180,E1 -2926.803,E2 -2926.803} C_VEL
LIN {X 0,Y 559.157,Z 87.144,A -85,B 0,C 180,E1 -2929.187,E2 -2929.187} C_VEL
LIN {X 0,Y 559.134,Z 87.153,A -85,B 0,C 180,E1 -2931.982,E2 -2931.982} C_VEL
LIN {X 0,Y 559.133,Z 87.148,A -85,B 0,C 180,E1 -2934.787,E2 -2934.787} C_VEL
LIN {X 0,Y 559.175,Z 87.151,A -85,B 0,C 180,E1 -2937.361,E2 -2937.361} C_VEL
LIN {X 0,Y 559.171,Z 87.281,A -85,B 0,C 180,E1 -2940.054,E2 -2940.054} C_VEL
LIN {X 0,Y 562.212,Z 97.689,A -85,B 0,C 180,E1 -2941.05,E2 -2941.05} C_VEL
LIN {X 0,Y 562.013,Z 120.057,A -85,B 0,C 180,E1 -2942.833,E2 -2942.833} C_VEL
LIN {X 0,Y 561.604,Z 155.53,A -85,B 0,C 180,E1 -2945.608,E2 -2945.608} C_VEL
LIN {X 0,Y 561.607,Z 157.462,A -85,B 0,C 180,E1 -2945.735,E2 -2945.735} C_VEL
LIN {X 0,Y 563.162,Z 167.209,A -85,B 0,C 180,E1 -2945.936,E2 -2945.936} C_VEL
LIN {X 0,Y 562.256,Z 366.361,A -85,B 0,C 180,E1 -2948.602,E2 -2948.602} C_VEL
LIN {X 0,Y 562.06,Z 382.988,A -85,B 0,C 180,E1 -2948.979,E2 -2948.979} C_VEL
LIN {X 0,Y 561.743,Z 399.225,A -85,B 0,C 180,E1 -2949.493,E2 -2949.493} C_VEL
LIN {X 0,Y 561.429,Z 415.532,A -85,B 0,C 180,E1 -2950.172,E2 -2950.172} C_VEL
LIN {X 0,Y 561.096,Z 429.7,A -85,B 0,C 180,E1 -2950.899,E2 -2950.899} C_VEL
LIN {X 0,Y 560.706,Z 444.681,A -85,B 0,C 180,E1 -2951.833,E2 -2951.833} C_VEL
LIN {X 0,Y 560.266,Z 459.547,A -85,B 0,C 180,E1 -2952.949,E2 -2952.949} C_VEL
LIN {X 0,Y 559.953,Z 473.011,A -85,B 0,C 180,E1 -2954.158,E2 -2954.158} C_VEL
LIN {X 0,Y 559.626,Z 485.256,A -85,B 0,C 180,E1 -2955.453,E2 -2955.453} C_VEL
LIN {X 0,Y 559.4,Z 495.695,A -85,B 0,C 180,E1 -2956.745,E2 -2956.745} C_VEL
LIN {X 0,Y 559.201,Z 505.811,A -85,B 0,C 180,E1 -2958.215,E2 -2958.215} C_VEL
LIN {X 0,Y 559.067,Z 513.28,A -85,B 0,C 180,E1 -2959.497,E2 -2959.497} C_VEL
LIN {X 0,Y 558.938,Z 520.488,A -85,B 0,C 180,E1 -2960.957,E2 -2960.957} C_VEL
LIN {X 0,Y 558.893,Z 526.464,A -85,B 0,C 180,E1 -2962.412,E2 -2962.412} C_VEL
LIN {X 0,Y 558.865,Z 532.247,A -85,B 0,C 180,E1 -2964.226,E2 -2964.226} C_VEL
LIN {X 0,Y 558.805,Z 535.635,A -85,B 0,C 180,E1 -2965.672,E2 -2965.672} C_VEL
LIN {X 0,Y 558.789,Z 538.089,A -85,B 0,C 180,E1 -2967.116,E2 -2967.116} C_VEL
LIN {X 0,Y 558.742,Z 539.479,A -85,B 0,C 180,E1 -2968.558,E2 -2968.558} C_VEL
LIN {X 0,Y 558.735,Z 540,A -85,B 0,C 180,E1 -2970,E2 -2970} C_VEL
LIN {X 0,Y 558.742,Z 539.479,A -85,B 0,C 180,E1 -2971.441,E2 -2971.441} C_VEL
LIN {X 0,Y 558.788,Z 538.089,A -85,B 0,C 180,E1 -2972.883,E2 -2972.883} C_VEL
LIN {X 0,Y 558.804,Z 535.636,A -85,B 0,C 180,E1 -2974.327,E2 -2974.327} C_VEL
LIN {X 0,Y 558.864,Z 532.252,A -85,B 0,C 180,E1 -2975.773,E2 -2975.773} C_VEL
LIN {X 0,Y 558.894,Z 526.47,A -85,B 0,C 180,E1 -2977.587,E2 -2977.587} C_VEL
LIN {X 0,Y 558.94,Z 518.859,A -85,B 0,C 180,E1 -2979.407,E2 -2979.407} C_VEL
LIN {X 0,Y 559.115,Z 510.285,A -85,B 0,C 180,E1 -2981.046,E2 -2981.046} C_VEL
LIN {X 0,Y 559.275,Z 500.981,A -85,B 0,C 180,E1 -2982.519,E2 -2982.519} C_VEL
LIN {X 0,Y 559.47,Z 491.425,A -85,B 0,C 180,E1 -2983.808,E2 -2983.808} C_VEL
LIN {X 0,Y 559.79,Z 480.265,A -85,B 0,C 180,E1 -2985.102,E2 -2985.102} C_VEL
LIN {X 0,Y 560.049,Z 468.144,A -85,B 0,C 180,E1 -2986.306,E2 -2986.306} C_VEL
LIN {X 0,Y 560.419,Z 454.872,A -85,B 0,C 180,E1 -2987.421,E2 -2987.421} C_VEL
LIN {X 0,Y 560.806,Z 440.424,A -85,B 0,C 180,E1 -2988.447,E2 -2988.447} C_VEL
LIN {X 0,Y 561.192,Z 426.28,A -85,B 0,C 180,E1 -2989.287,E2 -2989.287} C_VEL
LIN {X 0,Y 561.539,Z 411.588,A -85,B 0,C 180,E1 -2990.012,E2 -2990.012} C_VEL
LIN {X 0,Y 561.857,Z 395.355,A -85,B 0,C 180,E1 -2990.645,E2 -2990.645} C_VEL
LIN {X 0,Y 562.138,Z 379.369,A -85,B 0,C 180,E1 -2991.113,E2 -2991.113} C_VEL
LIN {X 0,Y 562.284,Z 363.401,A -85,B 0,C 180,E1 -2991.444,E2 -2991.444} C_VEL
LIN {X 0,Y 563.125,Z 166.79,A -85,B 0,C 180,E1 -2994.068,E2 -2994.068} C_VEL
LIN {X 0,Y 561.724,Z 157.693,A -85,B 0,C 180,E1 -2994.279,E2 -2994.279} C_VEL
LIN {X 0,Y 562.372,Z 119.751,A -85,B 0,C 180,E1 -2997.305,E2 -2997.305} C_VEL
LIN {X 0,Y 562.664,Z 98.496,A -85,B 0,C 180,E1 -2999.033,E2 -2999.033} C_VEL
LIN {X 0,Y 559.189,Z 87.146,A -85,B 0,C 180,E1 -3000.18,E2 -3000.18} C_VEL
LIN {X 0,Y 559.173,Z 87.149,A -85,B 0,C 180,E1 -3002.713,E2 -3002.713} C_VEL
LIN {X 0,Y 559.126,Z 87.147,A -85,B 0,C 180,E1 -3005.323,E2 -3005.323} C_VEL
LIN {X 0,Y 559.128,Z 87.148,A -85,B 0,C 180,E1 -3008.017,E2 -3008.017} C_VEL
LIN {X 0,Y 559.155,Z 87.147,A -85,B 0,C 180,E1 -3010.812,E2 -3010.812} C_VEL
LIN {X 0,Y 559.159,Z 87.142,A -85,B 0,C 180,E1 -3013.731,E2 -3013.731} C_VEL
LIN {X 0,Y 559.142,Z 87.146,A -85,B 0,C 180,E1 -3016.803,E2 -3016.803} C_VEL
LIN {X 0,Y 559.169,Z 87.14,A -85,B 0,C 180,E1 -3019.189,E2 -3019.189} C_VEL
LIN {X 0,Y 559.131,Z 87.149,A -85,B 0,C 180,E1 -3021.982,E2 -3021.982} C_VEL
LIN {X 0,Y 559.154,Z 87.143,A -85,B 0,C 180,E1 -3024.783,E2 -3024.783} C_VEL
LIN {X 0,Y 559.169,Z 87.14,A -85,B 0,C 180,E1 -3027.361,E2 -3027.361} C_VEL
LIN {X 0,Y 559.166,Z 87.15,A -85,B 0,C 180,E1 -3030.138,E2 -3030.138} C_VEL
LIN {X 0,Y 559.168,Z 87.14,A -85,B 0,C 180,E1 -3033.172,E2 -3033.172} C_VEL
LIN {X 0,Y 559.153,Z 87.143,A -85,B 0,C 180,E1 -3035.495,E2 -3035.495} C_VEL
LIN {X 0,Y 559.167,Z 87.141,A -85,B 0,C 180,E1 -3038.624,E2 -3038.624} C_VEL
LIN {X 0,Y 559.165,Z 87.14,A -85,B 0,C 180,E1 -3040.926,E2 -3040.926} C_VEL
LIN {X 0,Y 559.164,Z 87.149,A -85,B 0,C 180,E1 -3043.948,E2 -3043.948} C_VEL
LIN {X 0,Y 559.17,Z 87.144,A -85,B 0,C 180,E1 -3046.184,E2 -3046.184} C_VEL
LIN {X 0,Y 559.189,Z 87.138,A -85,B 0,C 180,E1 -3049.134,E2 -3049.134} C_VEL
LIN {X 0,Y 559.2,Z 87.141,A -85,B 0,C 180,E1 -3052.054,E2 -3052.054} C_VEL
LIN {X 0,Y 559.249,Z 87.13,A -85,B 0,C 180,E1 -3054.953,E2 -3054.953} C_VEL
LIN {X 0,Y 559.247,Z 87.137,A -85,B 0,C 180,E1 -3057.839,E2 -3057.839} C_VEL
LIN {X 0,Y 559.269,Z 87.127,A -85,B 0,C 180,E1 -3060.72,E2 -3060.72} C_VEL
LIN {X 0,Y 559.237,Z 87.132,A -85,B 0,C 180,E1 -3062.881,E2 -3062.881} C_VEL
LIN {X 0,Y 559.223,Z 87.138,A -85,B 0,C 180,E1 -3065.77,E2 -3065.77} C_VEL
LIN {X 0,Y 559.183,Z 87.138,A -85,B 0,C 180,E1 -3068.675,E2 -3068.675} C_VEL
LIN {X 0,Y 559.201,Z 87.142,A -85,B 0,C 180,E1 -3071.601,E2 -3071.601} C_VEL
LIN {X 0,Y 559.196,Z 87.136,A -85,B 0,C 180,E1 -3074.596,E2 -3074.596} C_VEL
LIN {X 0,Y 559.159,Z 87.147,A -85,B 0,C 180,E1 -3077.557,E2 -3077.557} C_VEL
LIN {X 0,Y 559.168,Z 87.141,A -85,B 0,C 180,E1 -3079.838,E2 -3079.838} C_VEL
LIN {X 0,Y 559.138,Z 87.143,A -85,B 0,C 180,E1 -3082.153,E2 -3082.153} C_VEL
LIN {X 0,Y 559.175,Z 87.149,A -85,B 0,C 180,E1 -3085.187,E2 -3085.187} C_VEL
LIN {X 0,Y 559.177,Z 87.14,A -85,B 0,C 180,E1 -3087.712,E2 -3087.712} C_VEL
LIN {X 0,Y 559.142,Z 87.146,A -85,B 0,C 180,E1 -3090.619,E2 -3090.619} C_VEL
LIN {X 0,Y 558.483,Z 87.234,A -85,B 0,C 180,E1 -3091.221,E2 -3091.221} C_VEL
LIN {X 0,Y 555.621,Z 87.59,A -85,B 0,C 180,E1 -3092.197,E2 -3092.197} C_VEL
LIN {X 0,Y 553.207,Z 87.891,A -85,B 0,C 180,E1 -3092.983,E2 -3092.983} C_VEL
LIN {X 0,Y 552.186,Z 88.011,A -85,B 0,C 180,E1 -3093.589,E2 -3093.589} C_VEL
LIN {X 0,Y 552.111,Z 88.019,A -85,B 0,C 180,E1 -3093.795,E2 -3093.795} C_VEL
LIN {X 0,Y 552.109,Z 88.025,A -85,B 0,C 180,E1 -3096.747,E2 -3096.747} C_VEL
LIN {X 0,Y 552.132,Z 88.018,A -85,B 0,C 180,E1 -3099.527,E2 -3099.527} C_VEL
LIN {X 0,Y 552.127,Z 88.019,A -85,B 0,C 180,E1 -3102.426,E2 -3102.426} C_VEL
LIN {X 0,Y 552.097,Z 88.021,A -85,B 0,C 180,E1 -3105.563,E2 -3105.563} C_VEL
LIN {X 0,Y 552.138,Z 88.023,A -85,B 0,C 180,E1 -3108.676,E2 -3108.676} C_VEL
LIN {X 0,Y 552.117,Z 88.019,A -85,B 0,C 180,E1 -3111.412,E2 -3111.412} C_VEL
LIN {X 0,Y 552.083,Z 88.024,A -85,B 0,C 180,E1 -3114.157,E2 -3114.157} C_VEL
LIN {X 0,Y 552.121,Z 88.024,A -85,B 0,C 180,E1 -3116.815,E2 -3116.815} C_VEL
LIN {X 0,Y 552.104,Z 88.02,A -85,B 0,C 180,E1 -3119.391,E2 -3119.391} C_VEL
LIN {X 0,Y 552.118,Z 88.019,A -85,B 0,C 180,E1 -3121.903,E2 -3121.903} C_VEL
LIN {X 0,Y 552.154,Z 88.021,A -85,B 0,C 180,E1 -3124.65,E2 -3124.65} C_VEL
LIN {X 0,Y 552.092,Z 88.021,A -85,B 0,C 180,E1 -3127.55,E2 -3127.55} C_VEL
LIN {X 0,Y 552.148,Z 88.024,A -85,B 0,C 180,E1 -3130.374,E2 -3130.374} C_VEL
LIN {X 0,Y 552.155,Z 88.015,A -85,B 0,C 180,E1 -3132.978,E2 -3132.978} C_VEL
LIN {X 0,Y 552.135,Z 88.021,A -85,B 0,C 180,E1 -3136.005,E2 -3136.005} C_VEL
LIN {X 0,Y 552.163,Z 88.013,A -85,B 0,C 180,E1 -3138.994,E2 -3138.994} C_VEL
LIN {X 0,Y 552.158,Z 88.018,A -85,B 0,C 180,E1 -3141.952,E2 -3141.952} C_VEL
LIN {X 0,Y 552.227,Z 88.005,A -85,B 0,C 180,E1 -3144.889,E2 -3144.889} C_VEL
LIN {X 0,Y 552.225,Z 88.009,A -85,B 0,C 180,E1 -3147.812,E2 -3147.812} C_VEL
LIN {X 0,Y 552.243,Z 88.003,A -85,B 0,C 180,E1 -3150.73,E2 -3150.73} C_VEL
LIN {X 0,Y 552.204,Z 88.007,A -85,B 0,C 180,E1 -3152.919,E2 -3152.919} C_VEL
LIN {X 0,Y 552.199,Z 88.016,A -85,B 0,C 180,E1 -3155.844,E2 -3155.844} C_VEL
LIN {X 0,Y 552.159,Z 88.013,A -85,B 0,C 180,E1 -3158.786,E2 -3158.786} C_VEL
LIN {X 0,Y 552.164,Z 88.02,A -85,B 0,C 180,E1 -3161.751,E2 -3161.751} C_VEL
LIN {X 0,Y 552.138,Z 88.015,A -85,B 0,C 180,E1 -3164.749,E2 -3164.749} C_VEL
LIN {X 0,Y 552.111,Z 88.028,A -85,B 0,C 180,E1 -3167.789,E2 -3167.789} C_VEL
LIN {X 0,Y 552.133,Z 88.02,A -85,B 0,C 180,E1 -3170.102,E2 -3170.102} C_VEL
LIN {X 0,Y 552.095,Z 88.021,A -85,B 0,C 180,E1 -3172.451,E2 -3172.451} C_VEL
LIN {X 0,Y 552.158,Z 88.018,A -85,B 0,C 180,E1 -3175.351,E2 -3175.351} C_VEL
LIN {X 0,Y 552.121,Z 88.02,A -85,B 0,C 180,E1 -3178.098,E2 -3178.098} C_VEL
LIN {X 0,Y 552.104,Z 88.019,A -85,B 0,C 180,E1 -3180.61,E2 -3180.61} C_VEL
LIN {X 0,Y 552.126,Z 88.022,A -85,B 0,C 180,E1 -3183.186,E2 -3183.186} C_VEL
LIN {X 0,Y 552.088,Z 88.025,A -85,B 0,C 180,E1 -3185.844,E2 -3185.844} C_VEL
LIN {X 0,Y 552.118,Z 88.018,A -85,B 0,C 180,E1 -3188.589,E2 -3188.589} C_VEL
LIN {X 0,Y 552.124,Z 88.025,A -85,B 0,C 180,E1 -3191.446,E2 -3191.446} C_VEL
LIN {X 0,Y 552.096,Z 88.021,A -85,B 0,C 180,E1 -3194.532,E2 -3194.532} C_VEL
LIN {X 0,Y 552.132,Z 88.02,A -85,B 0,C 180,E1 -3197.585,E2 -3197.585} C_VEL
LIN {X 0,Y 552.133,Z 88.017,A -85,B 0,C 180,E1 -3200.473,E2 -3200.473} C_VEL
LIN {X 0,Y 552.114,Z 88.026,A -85,B 0,C 180,E1 -3203.317,E2 -3203.317} C_VEL
LIN {X 0,Y 552.132,Z 88.017,A -85,B 0,C 180,E1 -3205.939,E2 -3205.939} C_VEL
LIN {X 0,Y 552.123,Z 88.021,A -85,B 0,C 180,E1 -3208.541,E2 -3208.541} C_VEL
LIN {X 0,Y 552.128,Z 88.022,A -85,B 0,C 180,E1 -3211.438,E2 -3211.438} C_VEL
LIN {X 0,Y 552.132,Z 88.022,A -85,B 0,C 180,E1 -3214.356,E2 -3214.356} C_VEL
LIN {X 0,Y 552.116,Z 88.026,A -85,B 0,C 180,E1 -3215.448,E2 -3215.448} C_VEL
LIN {X 0,Y 553.199,Z 91,A -85,B 0,C 180,E1 -3215.549,E2 -3215.549} C_VEL
LIN {X 0,Y 556.63,Z 98.39,A -85,B 0,C 180,E1 -3215.822,E2 -3215.822} C_VEL
LIN {X 0,Y 555.709,Z 267.455,A -85,B 0,C 180,E1 -3218.143,E2 -3218.143} C_VEL
LIN {X 0,Y 555.477,Z 290.634,A -85,B 0,C 180,E1 -3218.499,E2 -3218.499} C_VEL
LIN {X 0,Y 555.268,Z 306.985,A -85,B 0,C 180,E1 -3218.904,E2 -3218.904} C_VEL
LIN {X 0,Y 554.995,Z 322.967,A -85,B 0,C 180,E1 -3219.44,E2 -3219.44} C_VEL
LIN {X 0,Y 554.621,Z 337.824,A -85,B 0,C 180,E1 -3220.089,E2 -3220.089} C_VEL
LIN {X 0,Y 554.256,Z 352.032,A -85,B 0,C 180,E1 -3220.847,E2 -3220.847} C_VEL
LIN {X 0,Y 553.825,Z 366.681,A -85,B 0,C 180,E1 -3221.791,E2 -3221.791} C_VEL
LIN {X 0,Y 553.458,Z 379.113,A -85,B 0,C 180,E1 -3222.749,E2 -3222.749} C_VEL
LIN {X 0,Y 553.117,Z 388.558,A -85,B 0,C 180,E1 -3223.578,E2 -3223.578} C_VEL
LIN {X 0,Y 552.903,Z 398.036,A -85,B 0,C 180,E1 -3224.518,E2 -3224.518} C_VEL
LIN {X 0,Y 552.649,Z 406.451,A -85,B 0,C 180,E1 -3225.454,E2 -3225.454} C_VEL
LIN {X 0,Y 552.389,Z 415.324,A -85,B 0,C 180,E1 -3226.574,E2 -3226.574} C_VEL
LIN {X 0,Y 552.214,Z 423.11,A -85,B 0,C 180,E1 -3227.691,E2 -3227.691} C_VEL
LIN {X 0,Y 552.043,Z 430.965,A -85,B 0,C 180,E1 -3228.991,E2 -3228.991} C_VEL
LIN {X 0,Y 551.926,Z 436.8,A -85,B 0,C 180,E1 -3230.101,E2 -3230.101} C_VEL
LIN {X 0,Y 551.844,Z 441.886,A -85,B 0,C 180,E1 -3231.209,E2 -3231.209} C_VEL
LIN {X 0,Y 551.813,Z 447.53,A -85,B 0,C 180,E1 -3232.683,E2 -3232.683} C_VEL
LIN {X 0,Y 551.766,Z 450.159,A -85,B 0,C 180,E1 -3233.471,E2 -3233.471} C_VEL
LIN {X 0,Y 551.696,Z 453.975,A -85,B 0,C 180,E1 -3234.884,E2 -3234.884} C_VEL
LIN {X 0,Y 551.732,Z 456.881,A -85,B 0,C 180,E1 -3236.348,E2 -3236.348} C_VEL
LIN {X 0,Y 551.647,Z 458.825,A -85,B 0,C 180,E1 -3237.81,E2 -3237.81} C_VEL
LIN {X 0,Y 551.64,Z 459.798,A -85,B 0,C 180,E1 -3239.27,E2 -3239.27} C_VEL
LIN {X 0,Y 551.641,Z 459.826,A -85,B 0,C 180,E1 -3240.73,E2 -3240.73} C_VEL
LIN {X 0,Y 551.647,Z 458.909,A -85,B 0,C 180,E1 -3242.19,E2 -3242.19} C_VEL
LIN {X 0,Y 551.731,Z 457.019,A -85,B 0,C 180,E1 -3243.652,E2 -3243.652} C_VEL
LIN {X 0,Y 551.694,Z 454.169,A -85,B 0,C 180,E1 -3245.116,E2 -3245.116} C_VEL
LIN {X 0,Y 551.813,Z 449.09,A -85,B 0,C 180,E1 -3246.949,E2 -3246.949} C_VEL
LIN {X 0,Y 551.824,Z 443.764,A -85,B 0,C 180,E1 -3248.422,E2 -3248.422} C_VEL
LIN {X 0,Y 551.855,Z 439.009,A -85,B 0,C 180,E1 -3249.53,E2 -3249.53} C_VEL
LIN {X 0,Y 551.983,Z 432.495,A -85,B 0,C 180,E1 -3250.824,E2 -3250.824} C_VEL
LIN {X 0,Y 552.158,Z 424.868,A -85,B 0,C 180,E1 -3252.123,E2 -3252.123} C_VEL
LIN {X 0,Y 552.341,Z 417.328,A -85,B 0,C 180,E1 -3253.24,E2 -3253.24} C_VEL
LIN {X 0,Y 552.604,Z 408.727,A -85,B 0,C 180,E1 -3254.359,E2 -3254.359} C_VEL
LIN {X 0,Y 552.817,Z 400.613,A -85,B 0,C 180,E1 -3255.295,E2 -3255.295} C_VEL
LIN {X 0,Y 553.045,Z 391.47,A -85,B 0,C 180,E1 -3256.235,E2 -3256.235} C_VEL
LIN {X 0,Y 553.371,Z 381.249,A -85,B 0,C 180,E1 -3257.163,E2 -3257.163} C_VEL
LIN {X 0,Y 553.694,Z 370.827,A -85,B 0,C 180,E1 -3257.994,E2 -3257.994} C_VEL
LIN {X 0,Y 554.042,Z 359.557,A -85,B 0,C 180,E1 -3258.777,E2 -3258.777} C_VEL
LIN {X 0,Y 554.408,Z 345.144,A -85,B 0,C 180,E1 -3259.629,E2 -3259.629} C_VEL
LIN {X 0,Y 554.775,Z 329.452,A -85,B 0,C 180,E1 -3260.372,E2 -3260.372} C_VEL
LIN {X 0,Y 555.108,Z 314.013,A -85,B 0,C 180,E1 -3260.957,E2 -3260.957} C_VEL
LIN {X 0,Y 555.359,Z 296.781,A -85,B 0,C 180,E1 -3261.433,E2 -3261.433} C_VEL
LIN {X 0,Y 555.469,Z 281.571,A -85,B 0,C 180,E1 -3261.72,E2 -3261.72} C_VEL
LIN {X 0,Y 556.387,Z 130.213,A -85,B 0,C 180,E1 -3263.809,E2 -3263.809} C_VEL
LIN {X 0,Y 556.442,Z 98.136,A -85,B 0,C 180,E1 -3264.282,E2 -3264.282} C_VEL
LIN {X 0,Y 552.203,Z 88.892,A -85,B 0,C 180,E1 -3264.621,E2 -3264.621} C_VEL
LIN {X 0,Y 552.066,Z 88.033,A -85,B 0,C 180,E1 -3264.674,E2 -3264.674} C_VEL
LIN {X 0,Y 552.067,Z 88.033,A -85,B 0,C 180,E1 -3267.277,E2 -3267.277} C_VEL
LIN {X 0,Y 552.078,Z 88.027,A -85,B 0,C 180,E1 -3270.043,E2 -3270.043} C_VEL
LIN {X 0,Y 552.108,Z 88.028,A -85,B 0,C 180,E1 -3272.845,E2 -3272.845} C_VEL
LIN {X 0,Y 552.071,Z 88.027,A -85,B 0,C 180,E1 -3275.438,E2 -3275.438} C_VEL
LIN {X 0,Y 552.093,Z 88.025,A -85,B 0,C 180,E1 -3277.885,E2 -3277.885} C_VEL
LIN {X 0,Y 552.109,Z 88.028,A -85,B 0,C 180,E1 -3280.481,E2 -3280.481} C_VEL
LIN {X 0,Y 552.108,Z 88.022,A -85,B 0,C 180,E1 -3283.423,E2 -3283.423} C_VEL
LIN {X 0,Y 552.108,Z 88.023,A -85,B 0,C 180,E1 -3286.576,E2 -3286.576} C_VEL
LIN {X 0,Y 552.11,Z 88.025,A -85,B 0,C 180,E1 -3289.518,E2 -3289.518} C_VEL
LIN {X 0,Y 552.094,Z 88.026,A -85,B 0,C 180,E1 -3292.336,E2 -3292.336} C_VEL
LIN {X 0,Y 552.085,Z 88.028,A -85,B 0,C 180,E1 -3295.051,E2 -3295.051} C_VEL
LIN {X 0,Y 552.127,Z 88.03,A -85,B 0,C 180,E1 -3297.682,E2 -3297.682} C_VEL
LIN {X 0,Y 552.155,Z 88.19,A -85,B 0,C 180,E1 -3299.768,E2 -3299.768} C_VEL
LIN {X 0,Y 555.623,Z 100.455,A -85,B 0,C 180,E1 -3300.967,E2 -3300.967} C_VEL
LIN {X 0,Y 555.083,Z 135.911,A -85,B 0,C 180,E1 -3303.815,E2 -3303.815} C_VEL
LIN {X 0,Y 554.828,Z 156.472,A -85,B 0,C 180,E1 -3305.419,E2 -3305.419} C_VEL
LIN {X 0,Y 556.596,Z 167.662,A -85,B 0,C 180,E1 -3305.653,E2 -3305.653} C_VEL
LIN {X 0,Y 555.845,Z 288.491,A -85,B 0,C 180,E1 -3307.319,E2 -3307.319} C_VEL
LIN {X 0,Y 555.485,Z 365.793,A -85,B 0,C 180,E1 -3308.377,E2 -3308.377} C_VEL
LIN {X 0,Y 555.279,Z 382.807,A -85,B 0,C 180,E1 -3308.758,E2 -3308.758} C_VEL
LIN {X 0,Y 555.014,Z 398.073,A -85,B 0,C 180,E1 -3309.233,E2 -3309.233} C_VEL
LIN {X 0,Y 554.718,Z 413.874,A -85,B 0,C 180,E1 -3309.865,E2 -3309.865} C_VEL
LIN {X 0,Y 554.392,Z 427.959,A -85,B 0,C 180,E1 -3310.563,E2 -3310.563} C_VEL
LIN {X 0,Y 553.968,Z 441.833,A -85,B 0,C 180,E1 -3311.412,E2 -3311.412} C_VEL
LIN {X 0,Y 553.524,Z 456.126,A -85,B 0,C 180,E1 -3312.457,E2 -3312.457} C_VEL
LIN {X 0,Y 553.112,Z 469.109,A -85,B 0,C 180,E1 -3313.577,E2 -3313.577} C_VEL
LIN {X 0,Y 552.815,Z 480.439,A -85,B 0,C 180,E1 -3314.721,E2 -3314.721} C_VEL
LIN {X 0,Y 552.484,Z 491.416,A -85,B 0,C 180,E1 -3316.013,E2 -3316.013} C_VEL
LIN {X 0,Y 552.226,Z 502.204,A -85,B 0,C 180,E1 -3317.505,E2 -3317.505} C_VEL
LIN {X 0,Y 552.039,Z 511.265,A -85,B 0,C 180,E1 -3318.99,E2 -3318.99} C_VEL
LIN {X 0,Y 551.862,Z 518.853,A -85,B 0,C 180,E1 -3320.47,E2 -3320.47} C_VEL
LIN {X 0,Y 551.803,Z 526.464,A -85,B 0,C 180,E1 -3322.314,E2 -3322.314} C_VEL
LIN {X 0,Y 551.772,Z 532.247,A -85,B 0,C 180,E1 -3324.151,E2 -3324.151} C_VEL
LIN {X 0,Y 551.701,Z 535.634,A -85,B 0,C 180,E1 -3325.616,E2 -3325.616} C_VEL
LIN {X 0,Y 551.713,Z 538.09,A -85,B 0,C 180,E1 -3327.079,E2 -3327.079} C_VEL
LIN {X 0,Y 551.642,Z 539.479,A -85,B 0,C 180,E1 -3328.539,E2 -3328.539} C_VEL
LIN {X 0,Y 551.636,Z 540,A -85,B 0,C 180,E1 -3330,E2 -3330} C_VEL
LIN {X 0,Y 551.642,Z 539.479,A -85,B 0,C 180,E1 -3331.46,E2 -3331.46} C_VEL
LIN {X 0,Y 551.713,Z 538.09,A -85,B 0,C 180,E1 -3332.92,E2 -3332.92} C_VEL
LIN {X 0,Y 551.701,Z 535.635,A -85,B 0,C 180,E1 -3334.383,E2 -3334.383} C_VEL
LIN {X 0,Y 551.771,Z 532.253,A -85,B 0,C 180,E1 -3335.848,E2 -3335.848} C_VEL
LIN {X 0,Y 551.804,Z 526.469,A -85,B 0,C 180,E1 -3337.685,E2 -3337.685} C_VEL
LIN {X 0,Y 551.868,Z 518.858,A -85,B 0,C 180,E1 -3339.529,E2 -3339.529} C_VEL
LIN {X 0,Y 552.038,Z 511.27,A -85,B 0,C 180,E1 -3341.009,E2 -3341.009} C_VEL
LIN {X 0,Y 552.225,Z 502.212,A -85,B 0,C 180,E1 -3342.494,E2 -3342.494} C_VEL
LIN {X 0,Y 552.482,Z 491.425,A -85,B 0,C 180,E1 -3343.986,E2 -3343.986} C_VEL
LIN {X 0,Y 552.854,Z 480.453,A -85,B 0,C 180,E1 -3345.276,E2 -3345.276} C_VEL
LIN {X 0,Y 553.16,Z 468.143,A -85,B 0,C 180,E1 -3346.515,E2 -3346.515} C_VEL
LIN {X 0,Y 553.576,Z 454.639,A -85,B 0,C 180,E1 -3347.662,E2 -3347.662} C_VEL
LIN {X 0,Y 553.986,Z 440.42,A -85,B 0,C 180,E1 -3348.682,E2 -3348.682} C_VEL
LIN {X 0,Y 554.395,Z 426.168,A -85,B 0,C 180,E1 -3349.533,E2 -3349.533} C_VEL
LIN {X 0,Y 554.815,Z 410.942,A -85,B 0,C 180,E1 -3350.273,E2 -3350.273} C_VEL
LIN {X 0,Y 555.142,Z 394.508,A -85,B 0,C 180,E1 -3350.906,E2 -3350.906} C_VEL
LIN {X 0,Y 555.417,Z 378.918,A -85,B 0,C 180,E1 -3351.357,E2 -3351.357} C_VEL
LIN {X 0,Y 555.565,Z 362.681,A -85,B 0,C 180,E1 -3351.692,E2 -3351.692} C_VEL
LIN {X 0,Y 556.577,Z 168.38,A -85,B 0,C 180,E1 -3354.331,E2 -3354.331} C_VEL
LIN {X 0,Y 554.995,Z 157.464,A -85,B 0,C 180,E1 -3354.579,E2 -3354.579} C_VEL
LIN {X 0,Y 555.733,Z 120.594,A -85,B 0,C 180,E1 -3357.558,E2 -3357.558} C_VEL
LIN {X 0,Y 556.112,Z 101.39,A -85,B 0,C 180,E1 -3359.134,E2 -3359.134} C_VEL
LIN {X 0,Y 552.136,Z 88.025,A -85,B 0,C 180,E1 -3360.496,E2 -3360.496} C_VEL
LIN {X 0,Y 552.12,Z 88.023,A -85,B 0,C 180,E1 -3363.185,E2 -3363.185} C_VEL
LIN {X 0,Y 552.083,Z 88.025,A -85,B 0,C 180,E1 -3365.843,E2 -3365.843} C_VEL
LIN {X 0,Y 552.117,Z 88.022,A -85,B 0,C 180,E1 -3369.061,E2 -3369.061} C_VEL
LIN {X 0,Y 552.129,Z 88.018,A -85,B 0,C 180,E1 -3371.444,E2 -3371.444} C_VEL
LIN {X 0,Y 552.093,Z 88.03,A -85,B 0,C 180,E1 -3374.532,E2 -3374.532} C_VEL
LIN {X 0,Y 552.125,Z 88.017,A -85,B 0,C 180,E1 -3377.584,E2 -3377.584} C_VEL
LIN {X 0,Y 552.13,Z 88.023,A -85,B 0,C 180,E1 -3380.473,E2 -3380.473} C_VEL
LIN {X 0,Y 552.11,Z 88.019,A -85,B 0,C 180,E1 -3383.316,E2 -3383.316} C_VEL
LIN {X 0,Y 552.127,Z 88.022,A -85,B 0,C 180,E1 -3385.939,E2 -3385.939} C_VEL
LIN {X 0,Y 552.114,Z 88.022,A -85,B 0,C 180,E1 -3388.54,E2 -3388.54} C_VEL
LIN {X 0,Y 552.12,Z 88.018,A -85,B 0,C 180,E1 -3391.438,E2 -3391.438} C_VEL
LIN {X 0,Y 552.126,Z 88.022,A -85,B 0,C 180,E1 -3394.356,E2 -3394.356} C_VEL
LIN {X 0,Y 552.106,Z 88.02,A -85,B 0,C 180,E1 -3396.758,E2 -3396.758} C_VEL
LIN {X 0,Y 552.116,Z 88.018,A -85,B 0,C 180,E1 -3399.12,E2 -3399.12} C_VEL
LIN {X 0,Y 552.124,Z 88.019,A -85,B 0,C 180,E1 -3401.444,E2 -3401.444} C_VEL
LIN {X 0,Y 552.114,Z 88.025,A -85,B 0,C 180,E1 -3403.737,E2 -3403.737} C_VEL
LIN {X 0,Y 552.133,Z 88.024,A -85,B 0,C 180,E1 -3406.005,E2 -3406.005} C_VEL
LIN {X 0,Y 552.157,Z 88.013,A -85,B 0,C 180,E1 -3408.993,E2 -3408.993} C_VEL
LIN {X 0,Y 552.154,Z 88.02,A -85,B 0,C 180,E1 -3411.952,E2 -3411.952} C_VEL
LIN {X 0,Y 552.224,Z 88.005,A -85,B 0,C 180,E1 -3414.889,E2 -3414.889} C_VEL
LIN {X 0,Y 552.219,Z 88.013,A -85,B 0,C 180,E1 -3417.812,E2 -3417.812} C_VEL
LIN {X 0,Y 552.239,Z 88.003,A -85,B 0,C 180,E1 -3420.729,E2 -3420.729} C_VEL
LIN {X 0,Y 552.203,Z 88.008,A -85,B 0,C 180,E1 -3422.918,E2 -3422.918} C_VEL
LIN {X 0,Y 552.194,Z 88.013,A -85,B 0,C 180,E1 -3425.844,E2 -3425.844} C_VEL
LIN {X 0,Y 552.154,Z 88.014,A -85,B 0,C 180,E1 -3428.786,E2 -3428.786} C_VEL
LIN {X 0,Y 552.159,Z 88.017,A -85,B 0,C 180,E1 -3431.751,E2 -3431.751} C_VEL
LIN {X 0,Y 552.132,Z 88.017,A -85,B 0,C 180,E1 -3434.749,E2 -3434.749} C_VEL
LIN {X 0,Y 552.11,Z 88.022,A -85,B 0,C 180,E1 -3437.789,E2 -3437.789} C_VEL
LIN {X 0,Y 552.127,Z 88.017,A -85,B 0,C 180,E1 -3440.101,E2 -3440.101} C_VEL
LIN {X 0,Y 552.092,Z 88.021,A -85,B 0,C 180,E1 -3442.451,E2 -3442.451} C_VEL
LIN {X 0,Y 552.152,Z 88.021,A -85,B 0,C 180,E1 -3445.351,E2 -3445.351} C_VEL
LIN {X 0,Y 552.116,Z 88.018,A -85,B 0,C 180,E1 -3448.098,E2 -3448.098} C_VEL
LIN {X 0,Y 552.104,Z 88.022,A -85,B 0,C 180,E1 -3450.615,E2 -3450.615} C_VEL
LIN {X 0,Y 552.119,Z 88.025,A -85,B 0,C 180,E1 -3453.186,E2 -3453.186} C_VEL
LIN {X 0,Y 552.111,Z 88.019,A -85,B 0,C 180,E1 -3453.795,E2 -3453.795} C_VEL
LIN {X 0,Y 551.476,Z 88.1,A -85,B 0,C 180,E1 -3454.403,E2 -3454.403} C_VEL
LIN {X 0,Y 548.654,Z 88.458,A -85,B 0,C 180,E1 -3455.392,E2 -3455.392} C_VEL
LIN {X 0,Y 546.234,Z 88.763,A -85,B 0,C 180,E1 -3456.187,E2 -3456.187} C_VEL
LIN {X 0,Y 545.164,Z 88.894,A -85,B 0,C 180,E1 -3456.801,E2 -3456.801} C_VEL
LIN {X 0,Y 545.062,Z 88.904,A -85,B 0,C 180,E1 -3457.009,E2 -3457.009} C_VEL
LIN {X 0,Y 545.072,Z 88.896,A -85,B 0,C 180,E1 -3460.142,E2 -3460.142} C_VEL
LIN {X 0,Y 545.075,Z 88.901,A -85,B 0,C 180,E1 -3463.107,E2 -3463.107} C_VEL
LIN {X 0,Y 545.062,Z 88.898,A -85,B 0,C 180,E1 -3466.225,E2 -3466.225} C_VEL
LIN {X 0,Y 545.095,Z 88.901,A -85,B 0,C 180,E1 -3468.887,E2 -3468.887} C_VEL
LIN {X 0,Y 545.051,Z 88.898,A -85,B 0,C 180,E1 -3471.763,E2 -3471.763} C_VEL
LIN {X 0,Y 545.034,Z 88.907,A -85,B 0,C 180,E1 -3474.532,E2 -3474.532} C_VEL
LIN {X 0,Y 545.08,Z 88.896,A -85,B 0,C 180,E1 -3477.213,E2 -3477.213} C_VEL
LIN {X 0,Y 545.063,Z 88.897,A -85,B 0,C 180,E1 -3479.811,E2 -3479.811} C_VEL
LIN {X 0,Y 545.087,Z 88.9,A -85,B 0,C 180,E1 -3482.345,E2 -3482.345} C_VEL
LIN {X 0,Y 545.116,Z 88.895,A -85,B 0,C 180,E1 -3484.821,E2 -3484.821} C_VEL
LIN {X 0,Y 545.039,Z 88.9,A -85,B 0,C 180,E1 -3487.243,E2 -3487.243} C_VEL
LIN {X 0,Y 545.12,Z 88.899,A -85,B 0,C 180,E1 -3490.415,E2 -3490.415} C_VEL
LIN {X 0,Y 545.072,Z 88.896,A -85,B 0,C 180,E1 -3493.522,E2 -3493.522} C_VEL
LIN {X 0,Y 545.095,Z 88.895,A -85,B 0,C 180,E1 -3495.82,E2 -3495.82} C_VEL
LIN {X 0,Y 545.118,Z 88.891,A -85,B 0,C 180,E1 -3498.85,E2 -3498.85} C_VEL
LIN {X 0,Y 545.129,Z 88.893,A -85,B 0,C 180,E1 -3501.848,E2 -3501.848} C_VEL
LIN {X 0,Y 545.203,Z 88.88,A -85,B 0,C 180,E1 -3504.823,E2 -3504.823} C_VEL
LIN {X 0,Y 545.197,Z 88.885,A -85,B 0,C 180,E1 -3507.784,E2 -3507.784} C_VEL
LIN {X 0,Y 545.213,Z 88.879,A -85,B 0,C 180,E1 -3510.739,E2 -3510.739} C_VEL
LIN {X 0,Y 545.171,Z 88.883,A -85,B 0,C 180,E1 -3512.956,E2 -3512.956} C_VEL
LIN {X 0,Y 545.171,Z 88.892,A -85,B 0,C 180,E1 -3515.92,E2 -3515.92} C_VEL
LIN {X 0,Y 545.118,Z 88.89,A -85,B 0,C 180,E1 -3518.901,E2 -3518.901} C_VEL
LIN {X 0,Y 545.136,Z 88.896,A -85,B 0,C 180,E1 -3521.905,E2 -3521.905} C_VEL
LIN {X 0,Y 545.087,Z 88.894,A -85,B 0,C 180,E1 -3524.944,E2 -3524.944} C_VEL
LIN {X 0,Y 545.08,Z 88.9,A -85,B 0,C 180,E1 -3528.026,E2 -3528.026} C_VEL
LIN {X 0,Y 545.097,Z 88.893,A -85,B 0,C 180,E1 -3530.372,E2 -3530.372} C_VEL
LIN {X 0,Y 545.083,Z 88.902,A -85,B 0,C 180,E1 -3533.56,E2 -3533.56} C_VEL
LIN {X 0,Y 545.082,Z 88.898,A -85,B 0,C 180,E1 -3536.001,E2 -3536.001} C_VEL
LIN {X 0,Y 545.091,Z 88.893,A -85,B 0,C 180,E1 -3538.748,E2 -3538.748} C_VEL
LIN {X 0,Y 545.062,Z 88.904,A -85,B 0,C 180,E1 -3541.679,E2 -3541.679} C_VEL
LIN {X 0,Y 545.078,Z 88.895,A -85,B 0,C 180,E1 -3544.392,E2 -3544.392} C_VEL
LIN {X 0,Y 545.038,Z 88.908,A -85,B 0,C 180,E1 -3547.304,E2 -3547.304} C_VEL
LIN {X 0,Y 545.067,Z 88.897,A -85,B 0,C 180,E1 -3550.143,E2 -3550.143} C_VEL
LIN {X 0,Y 545.082,Z 88.901,A -85,B 0,C 180,E1 -3553.107,E2 -3553.107} C_VEL
LIN {X 0,Y 545.052,Z 88.898,A -85,B 0,C 180,E1 -3556.227,E2 -3556.227} C_VEL
LIN {X 0,Y 545.084,Z 88.899,A -85,B 0,C 180,E1 -3558.886,E2 -3558.886} C_VEL
LIN {X 0,Y 545.083,Z 88.898,A -85,B 0,C 180,E1 -3560.819,E2 -3560.819} C_VEL
LIN {X 0,Y 545.052,Z 88.902,A -85,B 0,C 180,E1 -3563.62,E2 -3563.62} C_VEL
LIN {X 0,Y 545.07,Z 88.897,A -85,B 0,C 180,E1 -3566.328,E2 -3566.328} C_VEL
LIN {X 0,Y 545.07,Z 88.905,A -85,B 0,C 180,E1 -3568.952,E2 -3568.952} C_VEL
LIN {X 0,Y 545.105,Z 88.897,A -85,B 0,C 180,E1 -3571.508,E2 -3571.508} C_VEL
LIN {X 0,Y 545.098,Z 88.9,A -85,B 0,C 180,E1 -3574.492,E2 -3574.492} C_VEL
LIN {X 0,Y 545.106,Z 89.029,A -85,B 0,C 180,E1 -3575.129,E2 -3575.129} C_VEL
LIN {X 0,Y 546.241,Z 91.976,A -85,B 0,C 180,E1 -3575.23,E2 -3575.23} C_VEL
LIN {X 0,Y 550.141,Z 100.368,A -85,B 0,C 180,E1 -3575.547,E2 -3575.547} C_VEL
LIN {X 0,Y 549.101,Z 258.747,A -85,B 0,C 180,E1 -3577.767,E2 -3577.767} C_VEL
LIN {X 0,Y 548.84,Z 289.643,A -85,B 0,C 180,E1 -3578.226,E2 -3578.226} C_VEL
LIN {X 0,Y 548.569,Z 306.411,A -85,B 0,C 180,E1 -3578.634,E2 -3578.634} C_VEL
LIN {X 0,Y 548.269,Z 322.533,A -85,B 0,C 180,E1 -3579.175,E2 -3579.175} C_VEL
LIN {X 0,Y 547.899,Z 337.653,A -85,B 0,C 180,E1 -3579.835,E2 -3579.835} C_VEL
LIN {X 0,Y 547.504,Z 351.945,A -85,B 0,C 180,E1 -3580.601,E2 -3580.601} C_VEL
LIN {X 0,Y 547.027,Z 366.711,A -85,B 0,C 180,E1 -3581.557,E2 -3581.557} C_VEL
LIN {X 0,Y 546.651,Z 378.512,A -85,B 0,C 180,E1 -3582.465,E2 -3582.465} C_VEL
LIN {X 0,Y 546.235,Z 388.707,A -85,B 0,C 180,E1 -3583.365,E2 -3583.365} C_VEL
LIN {X 0,Y 545.972,Z 398.172,A -85,B 0,C 180,E1 -3584.317,E2 -3584.317} C_VEL
LIN {X 0,Y 545.684,Z 406.543,A -85,B 0,C 180,E1 -3585.264,E2 -3585.264} C_VEL
LIN {X 0,Y 545.393,Z 415.338,A -85,B 0,C 180,E1 -3586.398,E2 -3586.398} C_VEL
LIN {X 0,Y 545.196,Z 423.103,A -85,B 0,C 180,E1 -3587.53,E2 -3587.53} C_VEL
LIN {X 0,Y 545.021,Z 430.96,A -85,B 0,C 180,E1 -3588.847,E2 -3588.847} C_VEL
LIN {X 0,Y 544.879,Z 436.795,A -85,B 0,C 180,E1 -3589.972,E2 -3589.972} C_VEL
LIN {X 0,Y 544.785,Z 441.879,A -85,B 0,C 180,E1 -3591.094,E2 -3591.094} C_VEL
LIN {X 0,Y 544.717,Z 447.527,A -85,B 0,C 180,E1 -3592.587,E2 -3592.587} C_VEL
LIN {X 0,Y 544.68,Z 450.436,A -85,B 0,C 180,E1 -3593.482,E2 -3593.482} C_VEL
LIN {X 0,Y 544.618,Z 453.968,A -85,B 0,C 180,E1 -3594.817,E2 -3594.817} C_VEL
LIN {X 0,Y 544.646,Z 456.878,A -85,B 0,C 180,E1 -3596.301,E2 -3596.301} C_VEL
LIN {X 0,Y 544.562,Z 458.818,A -85,B 0,C 180,E1 -3597.781,E2 -3597.781} C_VEL
LIN {X 0,Y 544.54,Z 459.792,A -85,B 0,C 180,E1 -3599.26,E2 -3599.26} C_VEL
LIN {X 0,Y 544.541,Z 459.819,A -85,B 0,C 180,E1 -3600.739,E2 -3600.739} C_VEL
LIN {X 0,Y 544.562,Z 458.901,A -85,B 0,C 180,E1 -3602.219,E2 -3602.219} C_VEL
LIN {X 0,Y 544.645,Z 457.015,A -85,B 0,C 180,E1 -3603.699,E2 -3603.699} C_VEL
LIN {X 0,Y 544.615,Z 454.159,A -85,B 0,C 180,E1 -3605.183,E2 -3605.183} C_VEL
LIN {X 0,Y 544.728,Z 449.083,A -85,B 0,C 180,E1 -3607.04,E2 -3607.04} C_VEL
LIN {X 0,Y 544.742,Z 443.752,A -85,B 0,C 180,E1 -3608.532,E2 -3608.532} C_VEL
LIN {X 0,Y 544.789,Z 438.998,A -85,B 0,C 180,E1 -3609.654,E2 -3609.654} C_VEL
LIN {X 0,Y 544.945,Z 432.484,A -85,B 0,C 180,E1 -3610.966,E2 -3610.966} C_VEL
LIN {X 0,Y 545.138,Z 424.853,A -85,B 0,C 180,E1 -3612.282,E2 -3612.282} C_VEL
LIN {X 0,Y 545.336,Z 417.316,A -85,B 0,C 180,E1 -3613.413,E2 -3613.413} C_VEL
LIN {X 0,Y 545.633,Z 408.825,A -85,B 0,C 180,E1 -3614.546,E2 -3614.546} C_VEL
LIN {X 0,Y 545.908,Z 400.767,A -85,B 0,C 180,E1 -3615.494,E2 -3615.494} C_VEL
LIN {X 0,Y 546.17,Z 391.645,A -85,B 0,C 180,E1 -3616.445,E2 -3616.445} C_VEL
LIN {X 0,Y 546.524,Z 381.552,A -85,B 0,C 180,E1 -3617.371,E2 -3617.371} C_VEL
LIN {X 0,Y 546.927,Z 369.732,A -85,B 0,C 180,E1 -3618.311,E2 -3618.311} C_VEL
LIN {X 0,Y 547.36,Z 354.941,A -85,B 0,C 180,E1 -3619.307,E2 -3619.307} C_VEL
LIN {X 0,Y 547.764,Z 341.114,A -85,B 0,C 180,E1 -3620.073,E2 -3620.073} C_VEL
LIN {X 0,Y 548.102,Z 326.917,A -85,B 0,C 180,E1 -3620.719,E2 -3620.719} C_VEL
LIN {X 0,Y 548.441,Z 309.946,A -85,B 0,C 180,E1 -3621.322,E2 -3621.322} C_VEL
LIN {X 0,Y 548.651,Z 294.063,A -85,B 0,C 180,E1 -3621.733,E2 -3621.733} C_VEL
LIN {X 0,Y 548.827,Z 277.127,A -85,B 0,C 180,E1 -3622.022,E2 -3622.022} C_VEL
LIN {X 0,Y 549.834,Z 131.321,A -85,B 0,C 180,E1 -3624.079,E2 -3624.079} C_VEL
LIN {X 0,Y 550.082,Z 100.442,A -85,B 0,C 180,E1 -3624.542,E2 -3624.542} C_VEL
LIN {X 0,Y 545.095,Z 89.4,A -85,B 0,C 180,E1 -3624.956,E2 -3624.956} C_VEL
LIN {X 0,Y 545.025,Z 88.911,A -85,B 0,C 180,E1 -3624.994,E2 -3624.994} C_VEL
LIN {X 0,Y 545.002,Z 88.91,A -85,B 0,C 180,E1 -3627.66,E2 -3627.66} C_VEL
LIN {X 0,Y 545.027,Z 88.907,A -85,B 0,C 180,E1 -3630.236,E2 -3630.236} C_VEL
LIN {X 0,Y 545.072,Z 88.902,A -85,B 0,C 180,E1 -3633.06,E2 -3633.06} C_VEL
LIN {X 0,Y 545.026,Z 88.905,A -85,B 0,C 180,E1 -3635.671,E2 -3635.671} C_VEL
LIN {X 0,Y 545.049,Z 88.907,A -85,B 0,C 180,E1 -3638.237,E2 -3638.237} C_VEL
LIN {X 0,Y 545.082,Z 88.897,A -85,B 0,C 180,E1 -3641.114,E2 -3641.114} C_VEL
LIN {X 0,Y 545.051,Z 88.907,A -85,B 0,C 180,E1 -3644.13,E2 -3644.13} C_VEL
LIN {X 0,Y 545.08,Z 88.897,A -85,B 0,C 180,E1 -3646.893,E2 -3646.893} C_VEL
LIN {X 0,Y 545.067,Z 88.906,A -85,B 0,C 180,E1 -3649.857,E2 -3649.857} C_VEL
LIN {X 0,Y 545.071,Z 88.9,A -85,B 0,C 180,E1 -3653.074,E2 -3653.074} C_VEL
LIN {X 0,Y 545.07,Z 88.905,A -85,B 0,C 180,E1 -3656.328,E2 -3656.328} C_VEL
LIN {X 0,Y 545.088,Z 89.046,A -85,B 0,C 180,E1 -3659.454,E2 -3659.454} C_VEL
LIN {X 0,Y 548.854,Z 101.969,A -85,B 0,C 180,E1 -3660.761,E2 -3660.761} C_VEL
LIN {X 0,Y 548.466,Z 129.733,A -85,B 0,C 180,E1 -3663.044,E2 -3663.044} C_VEL
LIN {X 0,Y 547.985,Z 155.207,A -85,B 0,C 180,E1 -3665.086,E2 -3665.086} C_VEL
LIN {X 0,Y 550.037,Z 169.742,A -85,B 0,C 180,E1 -3665.397,E2 -3665.397} C_VEL
LIN {X 0,Y 549.054,Z 308.286,A -85,B 0,C 180,E1 -3667.359,E2 -3667.359} C_VEL
LIN {X 0,Y 548.74,Z 364.971,A -85,B 0,C 180,E1 -3668.147,E2 -3668.147} C_VEL
LIN {X 0,Y 548.456,Z 381.975,A -85,B 0,C 180,E1 -3668.53,E2 -3668.53} C_VEL
LIN {X 0,Y 548.172,Z 398.277,A -85,B 0,C 180,E1 -3669.048,E2 -3669.048} C_VEL
LIN {X 0,Y 547.789,Z 414.87,A -85,B 0,C 180,E1 -3669.732,E2 -3669.732} C_VEL
LIN {X 0,Y 547.424,Z 429.848,A -85,B 0,C 180,E1 -3670.5,E2 -3670.5} C_VEL
LIN {X 0,Y 546.978,Z 445.238,A -85,B 0,C 180,E1 -3671.457,E2 -3671.457} C_VEL
LIN {X 0,Y 546.519,Z 459.709,A -85,B 0,C 180,E1 -3672.54,E2 -3672.54} C_VEL
LIN {X 0,Y 546.155,Z 471.056,A -85,B 0,C 180,E1 -3673.554,E2 -3673.554} C_VEL
LIN {X 0,Y 545.806,Z 482.327,A -85,B 0,C 180,E1 -3674.732,E2 -3674.732} C_VEL
LIN {X 0,Y 545.467,Z 492.9,A -85,B 0,C 180,E1 -3676.02,E2 -3676.02} C_VEL
LIN {X 0,Y 545.229,Z 502.203,A -85,B 0,C 180,E1 -3677.342,E2 -3677.342} C_VEL
LIN {X 0,Y 545.017,Z 511.264,A -85,B 0,C 180,E1 -3678.847,E2 -3678.847} C_VEL
LIN {X 0,Y 544.796,Z 518.853,A -85,B 0,C 180,E1 -3680.345,E2 -3680.345} C_VEL
LIN {X 0,Y 544.739,Z 526.463,A -85,B 0,C 180,E1 -3682.214,E2 -3682.214} C_VEL
LIN {X 0,Y 544.688,Z 532.248,A -85,B 0,C 180,E1 -3684.075,E2 -3684.075} C_VEL
LIN {X 0,Y 544.599,Z 535.633,A -85,B 0,C 180,E1 -3685.559,E2 -3685.559} C_VEL
LIN {X 0,Y 544.639,Z 538.09,A -85,B 0,C 180,E1 -3687.041,E2 -3687.041} C_VEL
LIN {X 0,Y 544.543,Z 539.478,A -85,B 0,C 180,E1 -3688.52,E2 -3688.52} C_VEL
LIN {X 0,Y 544.536,Z 540,A -85,B 0,C 180,E1 -3690,E2 -3690} C_VEL
LIN {X 0,Y 544.543,Z 539.478,A -85,B 0,C 180,E1 -3691.479,E2 -3691.479} C_VEL
LIN {X 0,Y 544.639,Z 538.09,A -85,B 0,C 180,E1 -3692.958,E2 -3692.958} C_VEL
LIN {X 0,Y 544.599,Z 535.635,A -85,B 0,C 180,E1 -3694.44,E2 -3694.44} C_VEL
LIN {X 0,Y 544.687,Z 532.253,A -85,B 0,C 180,E1 -3695.924,E2 -3695.924} C_VEL
LIN {X 0,Y 544.738,Z 526.469,A -85,B 0,C 180,E1 -3697.785,E2 -3697.785} C_VEL
LIN {X 0,Y 544.801,Z 518.858,A -85,B 0,C 180,E1 -3699.654,E2 -3699.654} C_VEL
LIN {X 0,Y 545.015,Z 511.27,A -85,B 0,C 180,E1 -3701.152,E2 -3701.152} C_VEL
LIN {X 0,Y 545.228,Z 502.21,A -85,B 0,C 180,E1 -3702.657,E2 -3702.657} C_VEL
LIN {X 0,Y 545.528,Z 491.424,A -85,B 0,C 180,E1 -3704.168,E2 -3704.168} C_VEL
LIN {X 0,Y 545.925,Z 480.288,A -85,B 0,C 180,E1 -3705.493,E2 -3705.493} C_VEL
LIN {X 0,Y 546.262,Z 468.116,A -85,B 0,C 180,E1 -3706.73,E2 -3706.73} C_VEL
LIN {X 0,Y 546.676,Z 455.032,A -85,B 0,C 180,E1 -3707.833,E2 -3707.833} C_VEL
LIN {X 0,Y 547.07,Z 441.14,A -85,B 0,C 180,E1 -3708.83,E2 -3708.83} C_VEL
LIN {X 0,Y 547.511,Z 426.915,A -85,B 0,C 180,E1 -3709.691,E2 -3709.691} C_VEL
LIN {X 0,Y 547.98,Z 410.786,A -85,B 0,C 180,E1 -3710.492,E2 -3710.492} C_VEL
LIN {X 0,Y 548.37,Z 394.536,A -85,B 0,C 180,E1 -3711.128,E2 -3711.128} C_VEL
LIN {X 0,Y 548.665,Z 379.168,A -85,B 0,C 180,E1 -3711.583,E2 -3711.583} C_VEL
LIN {X 0,Y 548.862,Z 363.468,A -85,B 0,C 180,E1 -3711.921,E2 -3711.921} C_VEL
LIN {X 0,Y 549.267,Z 286.365,A -85,B 0,C 180,E1 -3712.984,E2 -3712.984} C_VEL
LIN {X 0,Y 550.024,Z 180.605,A -85,B 0,C 180,E1 -3714.454,E2 -3714.454} C_VEL
LIN {X 0,Y 549.952,Z 168.006,A -85,B 0,C 180,E1 -3714.643,E2 -3714.643} C_VEL
LIN {X 0,Y 548.288,Z 157.04,A -85,B 0,C 180,E1 -3714.903,E2 -3714.903} C_VEL
LIN {X 0,Y 549.096,Z 121.462,A -85,B 0,C 180,E1 -3717.815,E2 -3717.815} C_VEL
LIN {X 0,Y 549.475,Z 104.548,A -85,B 0,C 180,E1 -3719.22,E2 -3719.22} C_VEL
LIN {X 0,Y 549.046,Z 101.608,A -85,B 0,C 180,E1 -3719.492,E2 -3719.492} C_VEL
LIN {X 0,Y 545.078,Z 88.905,A -85,B 0,C 180,E1 -3720.823,E2 -3720.823} C_VEL
LIN {X 0,Y 545.066,Z 88.9,A -85,B 0,C 180,E1 -3723.671,E2 -3723.671} C_VEL
LIN {X 0,Y 545.066,Z 88.902,A -85,B 0,C 180,E1 -3726.926,E2 -3726.926} C_VEL
LIN {X 0,Y 545.062,Z 88.903,A -85,B 0,C 180,E1 -3730.142,E2 -3730.142} C_VEL
LIN {X 0,Y 545.083,Z 88.896,A -85,B 0,C 180,E1 -3733.105,E2 -3733.105} C_VEL
LIN {X 0,Y 545.052,Z 88.906,A -85,B 0,C 180,E1 -3736.225,E2 -3736.225} C_VEL
LIN {X 0,Y 545.087,Z 88.896,A -85,B 0,C 180,E1 -3738.886,E2 -3738.886} C_VEL
LIN {X 0,Y 545.05,Z 88.9,A -85,B 0,C 180,E1 -3741.763,E2 -3741.763} C_VEL
LIN {X 0,Y 545.06,Z 88.902,A -85,B 0,C 180,E1 -3744.534,E2 -3744.534} C_VEL
LIN {X 0,Y 545.077,Z 88.895,A -85,B 0,C 180,E1 -3747.212,E2 -3747.212} C_VEL
LIN {X 0,Y 545.098,Z 88.897,A -85,B 0,C 180,E1 -3749.813,E2 -3749.813} C_VEL
LIN {X 0,Y 545.089,Z 88.894,A -85,B 0,C 180,E1 -3752.826,E2 -3752.826} C_VEL
LIN {X 0,Y 545.048,Z 88.902,A -85,B 0,C 180,E1 -3755.631,E2 -3755.631} C_VEL
LIN {X 0,Y 545.061,Z 88.897,A -85,B 0,C 180,E1 -3758.837,E2 -3758.837} C_VEL
LIN {X 0,Y 545.078,Z 88.895,A -85,B 0,C 180,E1 -3761.196,E2 -3761.196} C_VEL
LIN {X 0,Y 545.07,Z 88.899,A -85,B 0,C 180,E1 -3763.521,E2 -3763.521} C_VEL
LIN {X 0,Y 545.092,Z 88.902,A -85,B 0,C 180,E1 -3765.82,E2 -3765.82} C_VEL
LIN {X 0,Y 545.113,Z 88.89,A -85,B 0,C 180,E1 -3768.849,E2 -3768.849} C_VEL
LIN {X 0,Y 545.124,Z 88.897,A -85,B 0,C 180,E1 -3771.847,E2 -3771.847} C_VEL
LIN {X 0,Y 545.2,Z 88.88,A -85,B 0,C 180,E1 -3774.823,E2 -3774.823} C_VEL
LIN {X 0,Y 545.191,Z 88.889,A -85,B 0,C 180,E1 -3777.784,E2 -3777.784} C_VEL
LIN {X 0,Y 545.209,Z 88.879,A -85,B 0,C 180,E1 -3780.739,E2 -3780.739} C_VEL
LIN {X 0,Y 545.169,Z 88.885,A -85,B 0,C 180,E1 -3782.956,E2 -3782.956} C_VEL
LIN {X 0,Y 545.166,Z 88.887,A -85,B 0,C 180,E1 -3785.92,E2 -3785.92} C_VEL
LIN {X 0,Y 545.113,Z 88.892,A -85,B 0,C 180,E1 -3788.9,E2 -3788.9} C_VEL
LIN {X 0,Y 545.131,Z 88.891,A -85,B 0,C 180,E1 -3791.904,E2 -3791.904} C_VEL
LIN {X 0,Y 545.082,Z 88.898,A -85,B 0,C 180,E1 -3794.944,E2 -3794.944} C_VEL
LIN {X 0,Y 545.078,Z 88.896,A -85,B 0,C 180,E1 -3798.026,E2 -3798.026} C_VEL
LIN {X 0,Y 545.091,Z 88.893,A -85,B 0,C 180,E1 -3800.372,E2 -3800.372} C_VEL
LIN {X 0,Y 545.088,Z 88.898,A -85,B 0,C 180,E1 -3803.559,E2 -3803.559} C_VEL
LIN {X 0,Y 545.076,Z 88.895,A -85,B 0,C 180,E1 -3806.001,E2 -3806.001} C_VEL
LIN {X 0,Y 545.085,Z 88.898,A -85,B 0,C 180,E1 -3808.749,E2 -3808.749} C_VEL
LIN {X 0,Y 545.074,Z 88.897,A -85,B 0,C 180,E1 -3811.683,E2 -3811.683} C_VEL
LIN {X 0,Y 545.078,Z 88.898,A -85,B 0,C 180,E1 -3814.563,E2 -3814.563} C_VEL
LIN {X 0,Y 545.062,Z 88.904,A -85,B 0,C 180,E1 -3817.009,E2 -3817.009} C_VEL
LIN {X 0,Y 544.355,Z 88.988,A -85,B 0,C 180,E1 -3817.625,E2 -3817.625} C_VEL
LIN {X 0,Y 541.491,Z 89.346,A -85,B 0,C 180,E1 -3818.626,E2 -3818.626} C_VEL
LIN {X 0,Y 539.105,Z 89.641,A -85,B 0,C 180,E1 -3819.432,E2 -3819.432} C_VEL
LIN {X 0,Y 538.095,Z 89.765,A -85,B 0,C 180,E1 -3820.054,E2 -3820.054} C_VEL
LIN {X 0,Y 538.019,Z 89.775,A -85,B 0,C 180,E1 -3820.265,E2 -3820.265} C_VEL
LIN {X 0,Y 538.023,Z 89.781,A -85,B 0,C 180,E1 -3822.988,E2 -3822.988} C_VEL
LIN {X 0,Y 538.026,Z 89.773,A -85,B 0,C 180,E1 -3825.926,E2 -3825.926} C_VEL
LIN {X 0,Y 538.049,Z 89.773,A -85,B 0,C 180,E1 -3829.225,E2 -3829.225} C_VEL
LIN {X 0,Y 537.99,Z 89.779,A -85,B 0,C 180,E1 -3832.123,E2 -3832.123} C_VEL
LIN {X 0,Y 537.996,Z 89.783,A -85,B 0,C 180,E1 -3834.916,E2 -3834.916} C_VEL
LIN {X 0,Y 538.025,Z 89.773,A -85,B 0,C 180,E1 -3837.618,E2 -3837.618} C_VEL
LIN {X 0,Y 538.016,Z 89.779,A -85,B 0,C 180,E1 -3840.239,E2 -3840.239} C_VEL
LIN {X 0,Y 538.062,Z 89.774,A -85,B 0,C 180,E1 -3842.797,E2 -3842.797} C_VEL
LIN {X 0,Y 538.048,Z 89.771,A -85,B 0,C 180,E1 -3845.293,E2 -3845.293} C_VEL
LIN {X 0,Y 538.014,Z 89.778,A -85,B 0,C 180,E1 -3848.042,E2 -3848.042} C_VEL
LIN {X 0,Y 538.036,Z 89.774,A -85,B 0,C 180,E1 -3850.941,E2 -3850.941} C_VEL
LIN {X 0,Y 538.023,Z 89.774,A -85,B 0,C 180,E1 -3853.3,E2 -3853.3} C_VEL
LIN {X 0,Y 538.064,Z 89.77,A -85,B 0,C 180,E1 -3855.631,E2 -3855.631} C_VEL
LIN {X 0,Y 538.078,Z 89.77,A -85,B 0,C 180,E1 -3858.702,E2 -3858.702} C_VEL
LIN {X 0,Y 538.086,Z 89.769,A -85,B 0,C 180,E1 -3861.74,E2 -3861.74} C_VEL
LIN {X 0,Y 538.161,Z 89.758,A -85,B 0,C 180,E1 -3864.755,E2 -3864.755} C_VEL
LIN {X 0,Y 538.169,Z 89.76,A -85,B 0,C 180,E1 -3867.755,E2 -3867.755} C_VEL
LIN {X 0,Y 538.183,Z 89.755,A -85,B 0,C 180,E1 -3870.749,E2 -3870.749} C_VEL
LIN {X 0,Y 538.138,Z 89.759,A -85,B 0,C 180,E1 -3872.995,E2 -3872.995} C_VEL
LIN {X 0,Y 538.124,Z 89.77,A -85,B 0,C 180,E1 -3875.998,E2 -3875.998} C_VEL
LIN {X 0,Y 538.069,Z 89.768,A -85,B 0,C 180,E1 -3879.018,E2 -3879.018} C_VEL
LIN {X 0,Y 538.085,Z 89.772,A -85,B 0,C 180,E1 -3882.063,E2 -3882.063} C_VEL
LIN {X 0,Y 538.047,Z 89.772,A -85,B 0,C 180,E1 -3885.144,E2 -3885.144} C_VEL
LIN {X 0,Y 538.032,Z 89.775,A -85,B 0,C 180,E1 -3888.271,E2 -3888.271} C_VEL
LIN {X 0,Y 538.041,Z 89.771,A -85,B 0,C 180,E1 -3890.652,E2 -3890.652} C_VEL
LIN {X 0,Y 538.006,Z 89.781,A -85,B 0,C 180,E1 -3893.889,E2 -3893.889} C_VEL
LIN {X 0,Y 538.044,Z 89.771,A -85,B 0,C 180,E1 -3896.367,E2 -3896.367} C_VEL
LIN {X 0,Y 538.033,Z 89.774,A -85,B 0,C 180,E1 -3898.934,E2 -3898.934} C_VEL
LIN {X 0,Y 538.017,Z 89.778,A -85,B 0,C 180,E1 -3901.888,E2 -3901.888} C_VEL
LIN {X 0,Y 538.014,Z 89.775,A -85,B 0,C 180,E1 -3904.618,E2 -3904.618} C_VEL
LIN {X 0,Y 538.006,Z 89.781,A -85,B 0,C 180,E1 -3907.17,E2 -3907.17} C_VEL
LIN {X 0,Y 538.024,Z 89.777,A -85,B 0,C 180,E1 -3909.797,E2 -3909.797} C_VEL
LIN {X 0,Y 538.022,Z 89.776,A -85,B 0,C 180,E1 -3912.786,E2 -3912.786} C_VEL
LIN {X 0,Y 538.022,Z 89.775,A -85,B 0,C 180,E1 -3915.927,E2 -3915.927} C_VEL
LIN {X 0,Y 538.033,Z 89.772,A -85,B 0,C 180,E1 -3918.227,E2 -3918.227} C_VEL
LIN {X 0,Y 538.016,Z 89.784,A -85,B 0,C 180,E1 -3921.17,E2 -3921.17} C_VEL
LIN {X 0,Y 538.005,Z 89.777,A -85,B 0,C 180,E1 -3924.088,E2 -3924.088} C_VEL
LIN {X 0,Y 538.034,Z 89.777,A -85,B 0,C 180,E1 -3926.728,E2 -3926.728} C_VEL
LIN {X 0,Y 538.03,Z 89.777,A -85,B 0,C 180,E1 -3929.556,E2 -3929.556} C_VEL
LIN {X 0,Y 538.044,Z 89.774,A -85,B 0,C 180,E1 -3931.95,E2 -3931.95} C_VEL
LIN {X 0,Y 538.078,Z 89.776,A -85,B 0,C 180,E1 -3934.779,E2 -3934.779} C_VEL
LIN {X 0,Y 539.26,Z 92.904,A -85,B 0,C 180,E1 -3934.9,E2 -3934.9} C_VEL
LIN {X 0,Y 543.656,Z 102.489,A -85,B 0,C 180,E1 -3935.267,E2 -3935.267} C_VEL
LIN {X 0,Y 542.409,Z 269.353,A -85,B 0,C 180,E1 -3937.653,E2 -3937.653} C_VEL
LIN {X 0,Y 542.147,Z 290.905,A -85,B 0,C 180,E1 -3937.993,E2 -3937.993} C_VEL
LIN {X 0,Y 541.89,Z 307.487,A -85,B 0,C 180,E1 -3938.407,E2 -3938.407} C_VEL
LIN {X 0,Y 541.559,Z 323.759,A -85,B 0,C 180,E1 -3938.968,E2 -3938.968} C_VEL
LIN {X 0,Y 541.114,Z 339.4,A -85,B 0,C 180,E1 -3939.67,E2 -3939.67} C_VEL
LIN {X 0,Y 540.689,Z 353.489,A -85,B 0,C 180,E1 -3940.445,E2 -3940.445} C_VEL
LIN {X 0,Y 540.166,Z 368.023,A -85,B 0,C 180,E1 -3941.412,E2 -3941.412} C_VEL
LIN {X 0,Y 539.789,Z 378.978,A -85,B 0,C 180,E1 -3942.266,E2 -3942.266} C_VEL
LIN {X 0,Y 539.317,Z 390.826,A -85,B 0,C 180,E1 -3943.34,E2 -3943.34} C_VEL
LIN {X 0,Y 538.93,Z 402.19,A -85,B 0,C 180,E1 -3944.533,E2 -3944.533} C_VEL
LIN {X 0,Y 538.553,Z 412.866,A -85,B 0,C 180,E1 -3945.837,E2 -3945.837} C_VEL
LIN {X 0,Y 538.216,Z 423.352,A -85,B 0,C 180,E1 -3947.366,E2 -3947.366} C_VEL
LIN {X 0,Y 537.983,Z 431.114,A -85,B 0,C 180,E1 -3948.699,E2 -3948.699} C_VEL
LIN {X 0,Y 537.838,Z 436.864,A -85,B 0,C 180,E1 -3949.839,E2 -3949.839} C_VEL
LIN {X 0,Y 537.73,Z 441.872,A -85,B 0,C 180,E1 -3950.977,E2 -3950.977} C_VEL
LIN {X 0,Y 537.639,Z 447.523,A -85,B 0,C 180,E1 -3952.489,E2 -3952.489} C_VEL
LIN {X 0,Y 537.6,Z 450.679,A -85,B 0,C 180,E1 -3953.487,E2 -3953.487} C_VEL
LIN {X 0,Y 537.543,Z 453.962,A -85,B 0,C 180,E1 -3954.749,E2 -3954.749} C_VEL
LIN {X 0,Y 537.562,Z 456.875,A -85,B 0,C 180,E1 -3956.252,E2 -3956.252} C_VEL
LIN {X 0,Y 537.482,Z 458.811,A -85,B 0,C 180,E1 -3957.752,E2 -3957.752} C_VEL
LIN {X 0,Y 537.44,Z 459.785,A -85,B 0,C 180,E1 -3959.251,E2 -3959.251} C_VEL
LIN {X 0,Y 537.438,Z 459.996,A -85,B 0,C 180,E1 -3960,E2 -3960} C_VEL
LIN {X 0,Y 537.444,Z 459.546,A -85,B 0,C 180,E1 -3961.499,E2 -3961.499} C_VEL
LIN {X 0,Y 537.544,Z 458.114,A -85,B 0,C 180,E1 -3962.998,E2 -3962.998} C_VEL
LIN {X 0,Y 537.499,Z 455.71,A -85,B 0,C 180,E1 -3964.5,E2 -3964.5} C_VEL
LIN {X 0,Y 537.578,Z 452.293,A -85,B 0,C 180,E1 -3966.003,E2 -3966.003} C_VEL
LIN {X 0,Y 537.645,Z 449.075,A -85,B 0,C 180,E1 -3967.133,E2 -3967.133} C_VEL
LIN {X 0,Y 537.676,Z 443.74,A -85,B 0,C 180,E1 -3968.645,E2 -3968.645} C_VEL
LIN {X 0,Y 537.83,Z 437.303,A -85,B 0,C 180,E1 -3970.161,E2 -3970.161} C_VEL
LIN {X 0,Y 538.057,Z 429.388,A -85,B 0,C 180,E1 -3971.725,E2 -3971.725} C_VEL
LIN {X 0,Y 538.312,Z 420.343,A -85,B 0,C 180,E1 -3973.207,E2 -3973.207} C_VEL
LIN {X 0,Y 538.666,Z 410.815,A -85,B 0,C 180,E1 -3974.526,E2 -3974.526} C_VEL
LIN {X 0,Y 539.017,Z 401.045,A -85,B 0,C 180,E1 -3975.697,E2 -3975.697} C_VEL
LIN {X 0,Y 539.377,Z 389.893,A -85,B 0,C 180,E1 -3976.853,E2 -3976.853} C_VEL
LIN {X 0,Y 539.859,Z 377.007,A -85,B 0,C 180,E1 -3977.991,E2 -3977.991} C_VEL
LIN {X 0,Y 540.3,Z 363.752,A -85,B 0,C 180,E1 -3978.977,E2 -3978.977} C_VEL
LIN {X 0,Y 540.74,Z 349.879,A -85,B 0,C 180,E1 -3979.849,E2 -3979.849} C_VEL
LIN {X 0,Y 541.244,Z 333.759,A -85,B 0,C 180,E1 -3980.67,E2 -3980.67} C_VEL
LIN {X 0,Y 541.574,Z 317.934,A -85,B 0,C 180,E1 -3981.306,E2 -3981.306} C_VEL
LIN {X 0,Y 541.84,Z 301.789,A -85,B 0,C 180,E1 -3981.795,E2 -3981.795} C_VEL
LIN {X 0,Y 542.001,Z 285.551,A -85,B 0,C 180,E1 -3982.138,E2 -3982.138} C_VEL
LIN {X 0,Y 543.269,Z 138.541,A -85,B 0,C 180,E1 -3984.264,E2 -3984.264} C_VEL
LIN {X 0,Y 543.46,Z 102.152,A -85,B 0,C 180,E1 -3984.832,E2 -3984.832} C_VEL
LIN {X 0,Y 538.148,Z 90.6,A -85,B 0,C 180,E1 -3985.296,E2 -3985.296} C_VEL
LIN {X 0,Y 537.98,Z 89.787,A -85,B 0,C 180,E1 -3985.325,E2 -3985.325} C_VEL
LIN {X 0,Y 537.976,Z 89.785,A -85,B 0,C 180,E1 -3988.053,E2 -3988.053} C_VEL
LIN {X 0,Y 537.996,Z 89.786,A -85,B 0,C 180,E1 -3990.628,E2 -3990.628} C_VEL
LIN {X 0,Y 538.021,Z 89.779,A -85,B 0,C 180,E1 -3993.278,E2 -3993.278} C_VEL
LIN {X 0,Y 537.991,Z 89.783,A -85,B 0,C 180,E1 -3996.005,E2 -3996.005} C_VEL
LIN {X 0,Y 538.011,Z 89.781,A -85,B 0,C 180,E1 -3998.83,E2 -3998.83} C_VEL
LIN {X 0,Y 538.031,Z 89.778,A -85,B 0,C 180,E1 -4001.773,E2 -4001.773} C_VEL
LIN {X 0,Y 538.008,Z 89.779,A -85,B 0,C 180,E1 -4004.862,E2 -4004.862} C_VEL
LIN {X 0,Y 538.02,Z 89.777,A -85,B 0,C 180,E1 -4007.214,E2 -4007.214} C_VEL
LIN {X 0,Y 538.024,Z 89.781,A -85,B 0,C 180,E1 -4010.203,E2 -4010.203} C_VEL
LIN {X 0,Y 538.025,Z 89.778,A -85,B 0,C 180,E1 -4013.067,E2 -4013.067} C_VEL
LIN {X 0,Y 538.021,Z 89.786,A -85,B 0,C 180,E1 -4015.826,E2 -4015.826} C_VEL
LIN {X 0,Y 538.031,Z 89.786,A -85,B 0,C 180,E1 -4018.938,E2 -4018.938} C_VEL
LIN {X 0,Y 538.048,Z 89.988,A -85,B 0,C 180,E1 -4019.13,E2 -4019.13} C_VEL
LIN {X 0,Y 542.204,Z 104.026,A -85,B 0,C 180,E1 -4020.598,E2 -4020.598} C_VEL
LIN {X 0,Y 541.743,Z 130.151,A -85,B 0,C 180,E1 -4022.787,E2 -4022.787} C_VEL
LIN {X 0,Y 541.223,Z 154.427,A -85,B 0,C 180,E1 -4024.764,E2 -4024.764} C_VEL
LIN {X 0,Y 543.489,Z 170.812,A -85,B 0,C 180,E1 -4025.129,E2 -4025.129} C_VEL
LIN {X 0,Y 542.301,Z 310.392,A -85,B 0,C 180,E1 -4027.146,E2 -4027.146} C_VEL
LIN {X 0,Y 541.95,Z 365.418,A -85,B 0,C 180,E1 -4027.934,E2 -4027.934} C_VEL
LIN {X 0,Y 541.651,Z 383.021,A -85,B 0,C 180,E1 -4028.347,E2 -4028.347} C_VEL
LIN {X 0,Y 541.251,Z 399.919,A -85,B 0,C 180,E1 -4028.908,E2 -4028.908} C_VEL
LIN {X 0,Y 540.891,Z 415.128,A -85,B 0,C 180,E1 -4029.561,E2 -4029.561} C_VEL
LIN {X 0,Y 540.48,Z 429.932,A -85,B 0,C 180,E1 -4030.338,E2 -4030.338} C_VEL
LIN {X 0,Y 540.034,Z 443.846,A -85,B 0,C 180,E1 -4031.21,E2 -4031.21} C_VEL
LIN {X 0,Y 539.568,Z 457.716,A -85,B 0,C 180,E1 -4032.251,E2 -4032.251} C_VEL
LIN {X 0,Y 539.187,Z 470.084,A -85,B 0,C 180,E1 -4033.336,E2 -4033.336} C_VEL
LIN {X 0,Y 538.839,Z 481.502,A -85,B 0,C 180,E1 -4034.491,E2 -4034.491} C_VEL
LIN {X 0,Y 538.477,Z 492.8,A -85,B 0,C 180,E1 -4035.834,E2 -4035.834} C_VEL
LIN {X 0,Y 538.206,Z 502.201,A -85,B 0,C 180,E1 -4037.174,E2 -4037.174} C_VEL
LIN {X 0,Y 537.98,Z 511.264,A -85,B 0,C 180,E1 -4038.699,E2 -4038.699} C_VEL
LIN {X 0,Y 537.74,Z 518.852,A -85,B 0,C 180,E1 -4040.217,E2 -4040.217} C_VEL
LIN {X 0,Y 537.658,Z 526.463,A -85,B 0,C 180,E1 -4042.111,E2 -4042.111} C_VEL
LIN {X 0,Y 537.588,Z 532.248,A -85,B 0,C 180,E1 -4043.996,E2 -4043.996} C_VEL
LIN {X 0,Y 537.5,Z 535.633,A -85,B 0,C 180,E1 -4045.5,E2 -4045.5} C_VEL
LIN {X 0,Y 537.539,Z 538.09,A -85,B 0,C 180,E1 -4047.002,E2 -4047.002} C_VEL
LIN {X 0,Y 537.448,Z 539.478,A -85,B 0,C 180,E1 -4048.501,E2 -4048.501} C_VEL
LIN {X 0,Y 537.437,Z 540,A -85,B 0,C 180,E1 -4050,E2 -4050} C_VEL
LIN {X 0,Y 537.448,Z 539.478,A -85,B 0,C 180,E1 -4051.498,E2 -4051.498} C_VEL
LIN {X 0,Y 537.539,Z 538.09,A -85,B 0,C 180,E1 -4052.997,E2 -4052.997} C_VEL
LIN {X 0,Y 537.499,Z 535.634,A -85,B 0,C 180,E1 -4054.499,E2 -4054.499} C_VEL
LIN {X 0,Y 537.587,Z 532.254,A -85,B 0,C 180,E1 -4056.003,E2 -4056.003} C_VEL
LIN {X 0,Y 537.658,Z 526.469,A -85,B 0,C 180,E1 -4057.888,E2 -4057.888} C_VEL
LIN {X 0,Y 537.743,Z 518.858,A -85,B 0,C 180,E1 -4059.782,E2 -4059.782} C_VEL
LIN {X 0,Y 537.989,Z 511.269,A -85,B 0,C 180,E1 -4061.3,E2 -4061.3} C_VEL
LIN {X 0,Y 538.205,Z 502.209,A -85,B 0,C 180,E1 -4062.825,E2 -4062.825} C_VEL
LIN {X 0,Y 538.479,Z 492.81,A -85,B 0,C 180,E1 -4064.165,E2 -4064.165} C_VEL
LIN {X 0,Y 538.894,Z 481.618,A -85,B 0,C 180,E1 -4065.506,E2 -4065.506} C_VEL
LIN {X 0,Y 539.242,Z 469.347,A -85,B 0,C 180,E1 -4066.759,E2 -4066.759} C_VEL
LIN {X 0,Y 539.677,Z 456.619,A -85,B 0,C 180,E1 -4067.873,E2 -4067.873} C_VEL
LIN {X 0,Y 540.121,Z 443.113,A -85,B 0,C 180,E1 -4068.885,E2 -4068.885} C_VEL
LIN {X 0,Y 540.625,Z 427.659,A -85,B 0,C 180,E1 -4069.853,E2 -4069.853} C_VEL
LIN {X 0,Y 541.147,Z 410.985,A -85,B 0,C 180,E1 -4070.7,E2 -4070.7} C_VEL
LIN {X 0,Y 541.555,Z 395.862,A -85,B 0,C 180,E1 -4071.307,E2 -4071.307} C_VEL
LIN {X 0,Y 541.931,Z 379.421,A -85,B 0,C 180,E1 -4071.815,E2 -4071.815} C_VEL
LIN {X 0,Y 542.184,Z 362.726,A -85,B 0,C 180,E1 -4072.18,E2 -4072.18} C_VEL
LIN {X 0,Y 542.583,Z 298.076,A -85,B 0,C 180,E1 -4073.089,E2 -4073.089} C_VEL
LIN {X 0,Y 543.42,Z 194.624,A -85,B 0,C 180,E1 -4074.556,E2 -4074.556} C_VEL
LIN {X 0,Y 543.495,Z 168.963,A -85,B 0,C 180,E1 -4074.935,E2 -4074.935} C_VEL
LIN {X 0,Y 541.599,Z 156.549,A -85,B 0,C 180,E1 -4075.239,E2 -4075.239} C_VEL
LIN {X 0,Y 542.504,Z 121.079,A -85,B 0,C 180,E1 -4078.183,E2 -4078.183} C_VEL
LIN {X 0,Y 542.86,Z 105.814,A -85,B 0,C 180,E1 -4079.469,E2 -4079.469} C_VEL
LIN {X 0,Y 539.355,Z 94.11,A -85,B 0,C 180,E1 -4080.683,E2 -4080.683} C_VEL
LIN {X 0,Y 538.037,Z 89.78,A -85,B 0,C 180,E1 -4081.17,E2 -4081.17} C_VEL
LIN {X 0,Y 538.02,Z 89.781,A -85,B 0,C 180,E1 -4084.172,E2 -4084.172} C_VEL
LIN {X 0,Y 538,Z 89.78,A -85,B 0,C 180,E1 -4087.17,E2 -4087.17} C_VEL
LIN {X 0,Y 538.019,Z 89.777,A -85,B 0,C 180,E1 -4089.797,E2 -4089.797} C_VEL
LIN {X 0,Y 538.02,Z 89.779,A -85,B 0,C 180,E1 -4092.785,E2 -4092.785} C_VEL
LIN {X 0,Y 538.028,Z 89.775,A -85,B 0,C 180,E1 -4095.14,E2 -4095.14} C_VEL
LIN {X 0,Y 538.03,Z 89.78,A -85,B 0,C 180,E1 -4098.227,E2 -4098.227} C_VEL
LIN {X 0,Y 538.012,Z 89.775,A -85,B 0,C 180,E1 -4101.17,E2 -4101.17} C_VEL
LIN {X 0,Y 538.025,Z 89.78,A -85,B 0,C 180,E1 -4104.083,E2 -4104.083} C_VEL
LIN {X 0,Y 538.027,Z 89.775,A -85,B 0,C 180,E1 -4106.727,E2 -4106.727} C_VEL
LIN {X 0,Y 538.033,Z 89.774,A -85,B 0,C 180,E1 -4109.554,E2 -4109.554} C_VEL
LIN {X 0,Y 538.04,Z 89.778,A -85,B 0,C 180,E1 -4111.95,E2 -4111.95} C_VEL
LIN {X 0,Y 538.067,Z 89.772,A -85,B 0,C 180,E1 -4114.467,E2 -4114.467} C_VEL
LIN {X 0,Y 538.019,Z 89.774,A -85,B 0,C 180,E1 -4116.928,E2 -4116.928} C_VEL
LIN {X 0,Y 538.075,Z 89.774,A -85,B 0,C 180,E1 -4120.148,E2 -4120.148} C_VEL
LIN {X 0,Y 538.021,Z 89.775,A -85,B 0,C 180,E1 -4123.299,E2 -4123.299} C_VEL
LIN {X 0,Y 538.06,Z 89.775,A -85,B 0,C 180,E1 -4125.631,E2 -4125.631} C_VEL
LIN {X 0,Y 538.072,Z 89.768,A -85,B 0,C 180,E1 -4128.702,E2 -4128.702} C_VEL
LIN {X 0,Y 538.081,Z 89.775,A -85,B 0,C 180,E1 -4131.74,E2 -4131.74} C_VEL
LIN {X 0,Y 538.157,Z 89.757,A -85,B 0,C 180,E1 -4134.755,E2 -4134.755} C_VEL
LIN {X 0,Y 538.163,Z 89.764,A -85,B 0,C 180,E1 -4137.755,E2 -4137.755} C_VEL
LIN {X 0,Y 538.179,Z 89.754,A -85,B 0,C 180,E1 -4140.748,E2 -4140.748} C_VEL
LIN {X 0,Y 538.136,Z 89.761,A -85,B 0,C 180,E1 -4142.995,E2 -4142.995} C_VEL
LIN {X 0,Y 538.119,Z 89.764,A -85,B 0,C 180,E1 -4145.997,E2 -4145.997} C_VEL
LIN {X 0,Y 538.064,Z 89.771,A -85,B 0,C 180,E1 -4149.018,E2 -4149.018} C_VEL
LIN {X 0,Y 538.079,Z 89.768,A -85,B 0,C 180,E1 -4152.063,E2 -4152.063} C_VEL
LIN {X 0,Y 538.041,Z 89.777,A -85,B 0,C 180,E1 -4155.144,E2 -4155.144} C_VEL
LIN {X 0,Y 538.03,Z 89.773,A -85,B 0,C 180,E1 -4158.27,E2 -4158.27} C_VEL
LIN {X 0,Y 538.036,Z 89.773,A -85,B 0,C 180,E1 -4160.652,E2 -4160.652} C_VEL
LIN {X 0,Y 538.021,Z 89.775,A -85,B 0,C 180,E1 -4163.888,E2 -4163.888} C_VEL
LIN {X 0,Y 538.038,Z 89.772,A -85,B 0,C 180,E1 -4166.367,E2 -4166.367} C_VEL
LIN {X 0,Y 538.027,Z 89.78,A -85,B 0,C 180,E1 -4168.934,E2 -4168.934} C_VEL
LIN {X 0,Y 538.024,Z 89.774,A -85,B 0,C 180,E1 -4171.891,E2 -4171.891} C_VEL
LIN {X 0,Y 538.028,Z 89.776,A -85,B 0,C 180,E1 -4174.621,E2 -4174.621} C_VEL
LIN {X 0,Y 538.005,Z 89.782,A -85,B 0,C 180,E1 -4177.171,E2 -4177.171} C_VEL
LIN {X 0,Y 538.019,Z 89.775,A -85,B 0,C 180,E1 -4180.265,E2 -4180.265} C_VEL
LIN {X 0,Y 537.368,Z 89.864,A -85,B 0,C 180,E1 -4180.89,E2 -4180.89} C_VEL
LIN {X 0,Y 534.518,Z 90.217,A -85,B 0,C 180,E1 -4181.905,E2 -4181.905} C_VEL
LIN {X 0,Y 532.094,Z 90.519,A -85,B 0,C 180,E1 -4182.722,E2 -4182.722} C_VEL
LIN {X 0,Y 531.047,Z 90.646,A -85,B 0,C 180,E1 -4183.353,E2 -4183.353} C_VEL
LIN {X 0,Y 530.959,Z 90.655,A -85,B 0,C 180,E1 -4183.567,E2 -4183.567} C_VEL
LIN {X 0,Y 530.964,Z 90.658,A -85,B 0,C 180,E1 -4186.506,E2 -4186.506} C_VEL
LIN {X 0,Y 530.987,Z 90.656,A -85,B 0,C 180,E1 -4188.976,E2 -4188.976} C_VEL
LIN {X 0,Y 530.956,Z 90.654,A -85,B 0,C 180,E1 -4191.53,E2 -4191.53} C_VEL
LIN {X 0,Y 530.951,Z 90.659,A -85,B 0,C 180,E1 -4194.38,E2 -4194.38} C_VEL
LIN {X 0,Y 530.969,Z 90.655,A -85,B 0,C 180,E1 -4197.134,E2 -4197.134} C_VEL
LIN {X 0,Y 530.968,Z 90.653,A -85,B 0,C 180,E1 -4199.804,E2 -4199.804} C_VEL
LIN {X 0,Y 531.013,Z 90.655,A -85,B 0,C 180,E1 -4202.467,E2 -4202.467} C_VEL
LIN {X 0,Y 531.005,Z 90.651,A -85,B 0,C 180,E1 -4204.943,E2 -4204.943} C_VEL
LIN {X 0,Y 530.97,Z 90.659,A -85,B 0,C 180,E1 -4208.247,E2 -4208.247} C_VEL
LIN {X 0,Y 530.995,Z 90.654,A -85,B 0,C 180,E1 -4210.678,E2 -4210.678} C_VEL
LIN {X 0,Y 530.985,Z 90.651,A -85,B 0,C 180,E1 -4213.072,E2 -4213.072} C_VEL
LIN {X 0,Y 531.019,Z 90.646,A -85,B 0,C 180,E1 -4215.436,E2 -4215.436} C_VEL
LIN {X 0,Y 531.037,Z 90.649,A -85,B 0,C 180,E1 -4218.55,E2 -4218.55} C_VEL
LIN {X 0,Y 531.055,Z 90.643,A -85,B 0,C 180,E1 -4221.63,E2 -4221.63} C_VEL
LIN {X 0,Y 531.12,Z 90.636,A -85,B 0,C 180,E1 -4224.686,E2 -4224.686} C_VEL
LIN {X 0,Y 531.14,Z 90.635,A -85,B 0,C 180,E1 -4227.726,E2 -4227.726} C_VEL
LIN {X 0,Y 531.153,Z 90.63,A -85,B 0,C 180,E1 -4230.759,E2 -4230.759} C_VEL
LIN {X 0,Y 531.105,Z 90.635,A -85,B 0,C 180,E1 -4233.035,E2 -4233.035} C_VEL
LIN {X 0,Y 531.084,Z 90.645,A -85,B 0,C 180,E1 -4236.078,E2 -4236.078} C_VEL
LIN {X 0,Y 531.03,Z 90.645,A -85,B 0,C 180,E1 -4239.139,E2 -4239.139} C_VEL
LIN {X 0,Y 531.042,Z 90.647,A -85,B 0,C 180,E1 -4242.225,E2 -4242.225} C_VEL
LIN {X 0,Y 530.997,Z 90.652,A -85,B 0,C 180,E1 -4245.35,E2 -4245.35} C_VEL
LIN {X 0,Y 530.991,Z 90.65,A -85,B 0,C 180,E1 -4248.522,E2 -4248.522} C_VEL
LIN {X 0,Y 531.002,Z 90.649,A -85,B 0,C 180,E1 -4250.938,E2 -4250.938} C_VEL
LIN {X 0,Y 530.968,Z 90.654,A -85,B 0,C 180,E1 -4254.226,E2 -4254.226} C_VEL
LIN {X 0,Y 531.006,Z 90.648,A -85,B 0,C 180,E1 -4256.744,E2 -4256.744} C_VEL
LIN {X 0,Y 530.984,Z 90.656,A -85,B 0,C 180,E1 -4259.323,E2 -4259.323} C_VEL
LIN {X 0,Y 530.973,Z 90.653,A -85,B 0,C 180,E1 -4262.101,E2 -4262.101} C_VEL
LIN {X 0,Y 530.973,Z 90.653,A -85,B 0,C 180,E1 -4264.851,E2 -4264.851} C_VEL
LIN {X 0,Y 530.967,Z 90.66,A -85,B 0,C 180,E1 -4267.508,E2 -4267.508} C_VEL
LIN {X 0,Y 530.983,Z 90.651,A -85,B 0,C 180,E1 -4270.433,E2 -4270.433} C_VEL
LIN {X 0,Y 530.962,Z 90.66,A -85,B 0,C 180,E1 -4273.495,E2 -4273.495} C_VEL
LIN {X 0,Y 530.957,Z 90.654,A -85,B 0,C 180,E1 -4276.505,E2 -4276.505} C_VEL
LIN {X 0,Y 530.987,Z 90.656,A -85,B 0,C 180,E1 -4278.977,E2 -4278.977} C_VEL
LIN {X 0,Y 530.96,Z 90.657,A -85,B 0,C 180,E1 -4281.53,E2 -4281.53} C_VEL
LIN {X 0,Y 530.966,Z 90.655,A -85,B 0,C 180,E1 -4284.381,E2 -4284.381} C_VEL
LIN {X 0,Y 530.97,Z 90.661,A -85,B 0,C 180,E1 -4287.134,E2 -4287.134} C_VEL
LIN {X 0,Y 530.973,Z 90.655,A -85,B 0,C 180,E1 -4289.803,E2 -4289.803} C_VEL
LIN {X 0,Y 531.016,Z 90.652,A -85,B 0,C 180,E1 -4292.468,E2 -4292.468} C_VEL
LIN {X 0,Y 531.037,Z 90.652,A -85,B 0,C 180,E1 -4294.435,E2 -4294.435} C_VEL
LIN {X 0,Y 532.17,Z 93.713,A -85,B 0,C 180,E1 -4294.553,E2 -4294.553} C_VEL
LIN {X 0,Y 537.214,Z 104.456,A -85,B 0,C 180,E1 -4294.979,E2 -4294.979} C_VEL
LIN {X 0,Y 535.708,Z 274.625,A -85,B 0,C 180,E1 -4297.46,E2 -4297.46} C_VEL
LIN {X 0,Y 535.486,Z 293.301,A -85,B 0,C 180,E1 -4297.781,E2 -4297.781} C_VEL
LIN {X 0,Y 535.183,Z 310.089,A -85,B 0,C 180,E1 -4298.224,E2 -4298.224} C_VEL
LIN {X 0,Y 534.81,Z 326.298,A -85,B 0,C 180,E1 -4298.813,E2 -4298.813} C_VEL
LIN {X 0,Y 534.351,Z 341.148,A -85,B 0,C 180,E1 -4299.501,E2 -4299.501} C_VEL
LIN {X 0,Y 533.842,Z 356.563,A -85,B 0,C 180,E1 -4300.384,E2 -4300.384} C_VEL
LIN {X 0,Y 533.272,Z 370.635,A -85,B 0,C 180,E1 -4301.362,E2 -4301.362} C_VEL
LIN {X 0,Y 532.796,Z 383.735,A -85,B 0,C 180,E1 -4302.438,E2 -4302.438} C_VEL
LIN {X 0,Y 532.242,Z 396.782,A -85,B 0,C 180,E1 -4303.704,E2 -4303.704} C_VEL
LIN {X 0,Y 531.785,Z 408.118,A -85,B 0,C 180,E1 -4305.007,E2 -4305.007} C_VEL
LIN {X 0,Y 531.441,Z 417.256,A -85,B 0,C 180,E1 -4306.229,E2 -4306.229} C_VEL
LIN {X 0,Y 531.156,Z 426.027,A -85,B 0,C 180,E1 -4307.584,E2 -4307.584} C_VEL
LIN {X 0,Y 530.912,Z 433.51,A -85,B 0,C 180,E1 -4308.934,E2 -4308.934} C_VEL
LIN {X 0,Y 530.714,Z 440.74,A -85,B 0,C 180,E1 -4310.472,E2 -4310.472} C_VEL
LIN {X 0,Y 530.599,Z 446.601,A -85,B 0,C 180,E1 -4312.006,E2 -4312.006} C_VEL
LIN {X 0,Y 530.526,Z 451.165,A -85,B 0,C 180,E1 -4313.487,E2 -4313.487} C_VEL
LIN {X 0,Y 530.468,Z 454.15,A -85,B 0,C 180,E1 -4314.679,E2 -4314.679} C_VEL
LIN {X 0,Y 530.481,Z 456.992,A -85,B 0,C 180,E1 -4316.202,E2 -4316.202} C_VEL
LIN {X 0,Y 530.403,Z 458.88,A -85,B 0,C 180,E1 -4317.722,E2 -4317.722} C_VEL
LIN {X 0,Y 530.342,Z 459.832,A -85,B 0,C 180,E1 -4319.241,E2 -4319.241} C_VEL
LIN {X 0,Y 530.339,Z 460.044,A -85,B 0,C 180,E1 -4320,E2 -4320} C_VEL
LIN {X 0,Y 530.354,Z 459.607,A -85,B 0,C 180,E1 -4321.519,E2 -4321.519} C_VEL
LIN {X 0,Y 530.449,Z 458.208,A -85,B 0,C 180,E1 -4323.038,E2 -4323.038} C_VEL
LIN {X 0,Y 530.405,Z 455.876,A -85,B 0,C 180,E1 -4324.56,E2 -4324.56} C_VEL
LIN {X 0,Y 530.508,Z 452.546,A -85,B 0,C 180,E1 -4326.084,E2 -4326.084} C_VEL
LIN {X 0,Y 530.579,Z 448.179,A -85,B 0,C 180,E1 -4327.612,E2 -4327.612} C_VEL
LIN {X 0,Y 530.656,Z 442.725,A -85,B 0,C 180,E1 -4329.145,E2 -4329.145} C_VEL
LIN {X 0,Y 530.877,Z 436.03,A -85,B 0,C 180,E1 -4330.681,E2 -4330.681} C_VEL
LIN {X 0,Y 531.125,Z 427.883,A -85,B 0,C 180,E1 -4332.223,E2 -4332.223} C_VEL
LIN {X 0,Y 531.392,Z 419.388,A -85,B 0,C 180,E1 -4333.577,E2 -4333.577} C_VEL
LIN {X 0,Y 531.762,Z 410.06,A -85,B 0,C 180,E1 -4334.86,E2 -4334.86} C_VEL
LIN {X 0,Y 532.164,Z 399.555,A -85,B 0,C 180,E1 -4336.101,E2 -4336.101} C_VEL
LIN {X 0,Y 532.695,Z 385.896,A -85,B 0,C 180,E1 -4337.466,E2 -4337.466} C_VEL
LIN {X 0,Y 533.173,Z 373.112,A -85,B 0,C 180,E1 -4338.542,E2 -4338.542} C_VEL
LIN {X 0,Y 533.682,Z 359.345,A -85,B 0,C 180,E1 -4339.521,E2 -4339.521} C_VEL
LIN {X 0,Y 534.176,Z 344.238,A -85,B 0,C 180,E1 -4340.405,E2 -4340.405} C_VEL
LIN {X 0,Y 534.572,Z 329.404,A -85,B 0,C 180,E1 -4341.108,E2 -4341.108} C_VEL
LIN {X 0,Y 534.959,Z 313.262,A -85,B 0,C 180,E1 -4341.709,E2 -4341.709} C_VEL
LIN {X 0,Y 535.204,Z 297.227,A -85,B 0,C 180,E1 -4342.155,E2 -4342.155} C_VEL
LIN {X 0,Y 535.38,Z 281.442,A -85,B 0,C 180,E1 -4342.452,E2 -4342.452} C_VEL
LIN {X 0,Y 536.562,Z 156.35,A -85,B 0,C 180,E1 -4344.294,E2 -4344.294} C_VEL
LIN {X 0,Y 537.066,Z 104.212,A -85,B 0,C 180,E1 -4345.124,E2 -4345.124} C_VEL
LIN {X 0,Y 531.107,Z 91.541,A -85,B 0,C 180,E1 -4345.663,E2 -4345.663} C_VEL
LIN {X 0,Y 530.935,Z 90.664,A -85,B 0,C 180,E1 -4345.704,E2 -4345.704} C_VEL
LIN {X 0,Y 530.933,Z 90.664,A -85,B 0,C 180,E1 -4348.459,E2 -4348.459} C_VEL
LIN {X 0,Y 530.942,Z 90.664,A -85,B 0,C 180,E1 -4351.08,E2 -4351.08} C_VEL
LIN {X 0,Y 530.957,Z 90.658,A -85,B 0,C 180,E1 -4353.775,E2 -4353.775} C_VEL
LIN {X 0,Y 530.952,Z 90.664,A -85,B 0,C 180,E1 -4356.559,E2 -4356.559} C_VEL
LIN {X 0,Y 530.971,Z 90.655,A -85,B 0,C 180,E1 -4359.444,E2 -4359.444} C_VEL
LIN {X 0,Y 530.979,Z 90.66,A -85,B 0,C 180,E1 -4362.456,E2 -4362.456} C_VEL
LIN {X 0,Y 530.983,Z 90.656,A -85,B 0,C 180,E1 -4365.621,E2 -4365.621} C_VEL
LIN {X 0,Y 530.995,Z 90.654,A -85,B 0,C 180,E1 -4368.564,E2 -4368.564} C_VEL
LIN {X 0,Y 530.958,Z 90.662,A -85,B 0,C 180,E1 -4371.529,E2 -4371.529} C_VEL
LIN {X 0,Y 530.955,Z 90.661,A -85,B 0,C 180,E1 -4374.38,E2 -4374.38} C_VEL
LIN {X 0,Y 530.972,Z 90.664,A -85,B 0,C 180,E1 -4377.133,E2 -4377.133} C_VEL
LIN {X 0,Y 530.975,Z 90.666,A -85,B 0,C 180,E1 -4378.755,E2 -4378.755} C_VEL
LIN {X 0,Y 535.651,Z 106.331,A -85,B 0,C 180,E1 -4380.443,E2 -4380.443} C_VEL
LIN {X 0,Y 534.861,Z 137.433,A -85,B 0,C 180,E1 -4383.085,E2 -4383.085} C_VEL
LIN {X 0,Y 534.512,Z 153.428,A -85,B 0,C 180,E1 -4384.413,E2 -4384.413} C_VEL
LIN {X 0,Y 536.992,Z 171.039,A -85,B 0,C 180,E1 -4384.831,E2 -4384.831} C_VEL
LIN {X 0,Y 535.652,Z 303.103,A -85,B 0,C 180,E1 -4386.8,E2 -4386.8} C_VEL
LIN {X 0,Y 535.219,Z 364.613,A -85,B 0,C 180,E1 -4387.693,E2 -4387.693} C_VEL
LIN {X 0,Y 534.858,Z 382.199,A -85,B 0,C 180,E1 -4388.108,E2 -4388.108} C_VEL
LIN {X 0,Y 534.477,Z 398.38,A -85,B 0,C 180,E1 -4388.649,E2 -4388.649} C_VEL
LIN {X 0,Y 534.038,Z 414.371,A -85,B 0,C 180,E1 -4389.337,E2 -4389.337} C_VEL
LIN {X 0,Y 533.561,Z 430.02,A -85,B 0,C 180,E1 -4390.173,E2 -4390.173} C_VEL
LIN {X 0,Y 533.082,Z 443.845,A -85,B 0,C 180,E1 -4391.055,E2 -4391.055} C_VEL
LIN {X 0,Y 532.549,Z 458.692,A -85,B 0,C 180,E1 -4392.19,E2 -4392.19} C_VEL
LIN {X 0,Y 532.07,Z 471.978,A -85,B 0,C 180,E1 -4393.402,E2 -4393.402} C_VEL
LIN {X 0,Y 531.7,Z 483.846,A -85,B 0,C 180,E1 -4394.671,E2 -4394.671} C_VEL
LIN {X 0,Y 531.359,Z 494.78,A -85,B 0,C 180,E1 -4396.031,E2 -4396.031} C_VEL
LIN {X 0,Y 531.09,Z 504.119,A -85,B 0,C 180,E1 -4397.388,E2 -4397.388} C_VEL
LIN {X 0,Y 530.847,Z 513.07,A -85,B 0,C 180,E1 -4398.932,E2 -4398.932} C_VEL
LIN {X 0,Y 530.648,Z 520.474,A -85,B 0,C 180,E1 -4400.47,E2 -4400.47} C_VEL
LIN {X 0,Y 530.569,Z 526.462,A -85,B 0,C 180,E1 -4402.005,E2 -4402.005} C_VEL
LIN {X 0,Y 530.496,Z 532.249,A -85,B 0,C 180,E1 -4403.916,E2 -4403.916} C_VEL
LIN {X 0,Y 530.403,Z 535.632,A -85,B 0,C 180,E1 -4405.44,E2 -4405.44} C_VEL
LIN {X 0,Y 530.444,Z 538.09,A -85,B 0,C 180,E1 -4406.962,E2 -4406.962} C_VEL
LIN {X 0,Y 530.358,Z 539.477,A -85,B 0,C 180,E1 -4408.481,E2 -4408.481} C_VEL
LIN {X 0,Y 530.338,Z 540,A -85,B 0,C 180,E1 -4409.999,E2 -4409.999} C_VEL
LIN {X 0,Y 530.358,Z 539.477,A -85,B 0,C 180,E1 -4411.518,E2 -4411.518} C_VEL
LIN {X 0,Y 530.444,Z 538.09,A -85,B 0,C 180,E1 -4413.037,E2 -4413.037} C_VEL
LIN {X 0,Y 530.403,Z 535.633,A -85,B 0,C 180,E1 -4414.559,E2 -4414.559} C_VEL
LIN {X 0,Y 530.495,Z 532.255,A -85,B 0,C 180,E1 -4416.083,E2 -4416.083} C_VEL
LIN {X 0,Y 530.568,Z 526.469,A -85,B 0,C 180,E1 -4417.994,E2 -4417.994} C_VEL
LIN {X 0,Y 530.653,Z 520.479,A -85,B 0,C 180,E1 -4419.529,E2 -4419.529} C_VEL
LIN {X 0,Y 530.849,Z 513.099,A -85,B 0,C 180,E1 -4421.067,E2 -4421.067} C_VEL
LIN {X 0,Y 531.088,Z 504.227,A -85,B 0,C 180,E1 -4422.611,E2 -4422.611} C_VEL
LIN {X 0,Y 531.421,Z 493.6,A -85,B 0,C 180,E1 -4424.161,E2 -4424.161} C_VEL
LIN {X 0,Y 531.881,Z 480.875,A -85,B 0,C 180,E1 -4425.716,E2 -4425.716} C_VEL
LIN {X 0,Y 532.24,Z 469.551,A -85,B 0,C 180,E1 -4426.887,E2 -4426.887} C_VEL
LIN {X 0,Y 532.736,Z 456.587,A -85,B 0,C 180,E1 -4428.045,E2 -4428.045} C_VEL
LIN {X 0,Y 533.201,Z 443.622,A -85,B 0,C 180,E1 -4429.039,E2 -4429.039} C_VEL
LIN {X 0,Y 533.745,Z 428.315,A -85,B 0,C 180,E1 -4430.02,E2 -4430.02} C_VEL
LIN {X 0,Y 534.257,Z 413.389,A -85,B 0,C 180,E1 -4430.804,E2 -4430.804} C_VEL
LIN {X 0,Y 534.719,Z 398.448,A -85,B 0,C 180,E1 -4431.444,E2 -4431.444} C_VEL
LIN {X 0,Y 535.132,Z 382.463,A -85,B 0,C 180,E1 -4431.98,E2 -4431.98} C_VEL
LIN {X 0,Y 535.455,Z 366.168,A -85,B 0,C 180,E1 -4432.372,E2 -4432.372} C_VEL
LIN {X 0,Y 535.854,Z 326.434,A -85,B 0,C 180,E1 -4432.965,E2 -4432.965} C_VEL
LIN {X 0,Y 536.325,Z 256.715,A -85,B 0,C 180,E1 -4433.967,E2 -4433.967} C_VEL
LIN {X 0,Y 537.129,Z 171.301,A -85,B 0,C 180,E1 -4435.207,E2 -4435.207} C_VEL
LIN {X 0,Y 534.925,Z 156.3,A -85,B 0,C 180,E1 -4435.564,E2 -4435.564} C_VEL
LIN {X 0,Y 535.891,Z 121.958,A -85,B 0,C 180,E1 -4438.453,E2 -4438.453} C_VEL
LIN {X 0,Y 536.301,Z 108.161,A -85,B 0,C 180,E1 -4439.627,E2 -4439.627} C_VEL
LIN {X 0,Y 533.099,Z 97.415,A -85,B 0,C 180,E1 -4440.757,E2 -4440.757} C_VEL
LIN {X 0,Y 530.983,Z 90.658,A -85,B 0,C 180,E1 -4441.492,E2 -4441.492} C_VEL
LIN {X 0,Y 530.986,Z 90.655,A -85,B 0,C 180,E1 -4443.772,E2 -4443.772} C_VEL
LIN {X 0,Y 530.951,Z 90.664,A -85,B 0,C 180,E1 -4446.558,E2 -4446.558} C_VEL
LIN {X 0,Y 530.982,Z 90.653,A -85,B 0,C 180,E1 -4449.443,E2 -4449.443} C_VEL
LIN {X 0,Y 530.978,Z 90.661,A -85,B 0,C 180,E1 -4452.456,E2 -4452.456} C_VEL
LIN {X 0,Y 530.981,Z 90.653,A -85,B 0,C 180,E1 -4455.621,E2 -4455.621} C_VEL
LIN {X 0,Y 530.992,Z 90.656,A -85,B 0,C 180,E1 -4458.564,E2 -4458.564} C_VEL
LIN {X 0,Y 530.955,Z 90.655,A -85,B 0,C 180,E1 -4461.529,E2 -4461.529} C_VEL
LIN {X 0,Y 530.977,Z 90.659,A -85,B 0,C 180,E1 -4464.382,E2 -4464.382} C_VEL
LIN {X 0,Y 530.966,Z 90.653,A -85,B 0,C 180,E1 -4467.134,E2 -4467.134} C_VEL
LIN {X 0,Y 530.98,Z 90.655,A -85,B 0,C 180,E1 -4469.804,E2 -4469.804} C_VEL
LIN {X 0,Y 531.011,Z 90.651,A -85,B 0,C 180,E1 -4472.467,E2 -4472.467} C_VEL
LIN {X 0,Y 531.002,Z 90.648,A -85,B 0,C 180,E1 -4474.942,E2 -4474.942} C_VEL
LIN {X 0,Y 530.967,Z 90.658,A -85,B 0,C 180,E1 -4478.247,E2 -4478.247} C_VEL
LIN {X 0,Y 530.992,Z 90.65,A -85,B 0,C 180,E1 -4480.677,E2 -4480.677} C_VEL
LIN {X 0,Y 530.982,Z 90.651,A -85,B 0,C 180,E1 -4483.071,E2 -4483.071} C_VEL
LIN {X 0,Y 531.015,Z 90.65,A -85,B 0,C 180,E1 -4485.436,E2 -4485.436} C_VEL
LIN {X 0,Y 531.044,Z 90.644,A -85,B 0,C 180,E1 -4488.55,E2 -4488.55} C_VEL
LIN {X 0,Y 531.051,Z 90.649,A -85,B 0,C 180,E1 -4491.63,E2 -4491.63} C_VEL
LIN {X 0,Y 531.117,Z 90.634,A -85,B 0,C 180,E1 -4494.685,E2 -4494.685} C_VEL
LIN {X 0,Y 531.135,Z 90.64,A -85,B 0,C 180,E1 -4497.725,E2 -4497.725} C_VEL
LIN {X 0,Y 531.149,Z 90.63,A -85,B 0,C 180,E1 -4500.758,E2 -4500.758} C_VEL
LIN {X 0,Y 531.102,Z 90.638,A -85,B 0,C 180,E1 -4503.034,E2 -4503.034} C_VEL
LIN {X 0,Y 531.079,Z 90.641,A -85,B 0,C 180,E1 -4506.077,E2 -4506.077} C_VEL
LIN {X 0,Y 531.024,Z 90.65,A -85,B 0,C 180,E1 -4509.138,E2 -4509.138} C_VEL
LIN {X 0,Y 531.037,Z 90.644,A -85,B 0,C 180,E1 -4512.225,E2 -4512.225} C_VEL
LIN {X 0,Y 530.992,Z 90.659,A -85,B 0,C 180,E1 -4515.35,E2 -4515.35} C_VEL
LIN {X 0,Y 530.988,Z 90.65,A -85,B 0,C 180,E1 -4518.521,E2 -4518.521} C_VEL
LIN {X 0,Y 530.996,Z 90.653,A -85,B 0,C 180,E1 -4520.938,E2 -4520.938} C_VEL
LIN {X 0,Y 530.976,Z 90.651,A -85,B 0,C 180,E1 -4524.225,E2 -4524.225} C_VEL
LIN {X 0,Y 531,Z 90.652,A -85,B 0,C 180,E1 -4526.744,E2 -4526.744} C_VEL
LIN {X 0,Y 530.978,Z 90.657,A -85,B 0,C 180,E1 -4529.323,E2 -4529.323} C_VEL
LIN {X 0,Y 530.976,Z 90.651,A -85,B 0,C 180,E1 -4532.103,E2 -4532.103} C_VEL
LIN {X 0,Y 530.985,Z 90.657,A -85,B 0,C 180,E1 -4534.854,E2 -4534.854} C_VEL
LIN {X 0,Y 530.963,Z 90.655,A -85,B 0,C 180,E1 -4537.508,E2 -4537.508} C_VEL
LIN {X 0,Y 530.982,Z 90.653,A -85,B 0,C 180,E1 -4540.433,E2 -4540.433} C_VEL
LIN {X 0,Y 530.963,Z 90.656,A -85,B 0,C 180,E1 -4543.282,E2 -4543.282} C_VEL
LIN {X 0,Y 530.959,Z 90.655,A -85,B 0,C 180,E1 -4543.567,E2 -4543.567} C_VEL
LIN {X 0,Y 530.287,Z 90.739,A -85,B 0,C 180,E1 -4544.2,E2 -4544.2} C_VEL
LIN {X 0,Y 527.441,Z 91.102,A -85,B 0,C 180,E1 -4545.229,E2 -4545.229} C_VEL
LIN {X 0,Y 525.039,Z 91.406,A -85,B 0,C 180,E1 -4546.058,E2 -4546.058} C_VEL
LIN {X 0,Y 524.006,Z 91.531,A -85,B 0,C 180,E1 -4546.697,E2 -4546.697} C_VEL
LIN {X 0,Y 523.92,Z 91.538,A -85,B 0,C 180,E1 -4546.914,E2 -4546.914} C_VEL
LIN {X 0,Y 523.945,Z 91.528,A -85,B 0,C 180,E1 -4549.921,E2 -4549.921} C_VEL
LIN {X 0,Y 523.904,Z 91.539,A -85,B 0,C 180,E1 -4552.868,E2 -4552.868} C_VEL
LIN {X 0,Y 523.93,Z 91.529,A -85,B 0,C 180,E1 -4555.71,E2 -4555.71} C_VEL
LIN {X 0,Y 523.922,Z 91.537,A -85,B 0,C 180,E1 -4558.457,E2 -4558.457} C_VEL
LIN {X 0,Y 523.937,Z 91.53,A -85,B 0,C 180,E1 -4561.126,E2 -4561.126} C_VEL
LIN {X 0,Y 523.983,Z 91.525,A -85,B 0,C 180,E1 -4563.981,E2 -4563.981} C_VEL
LIN {X 0,Y 523.935,Z 91.535,A -85,B 0,C 180,E1 -4566.271,E2 -4566.271} C_VEL
LIN {X 0,Y 523.945,Z 91.532,A -85,B 0,C 180,E1 -4568.767,E2 -4568.767} C_VEL
LIN {X 0,Y 523.951,Z 91.527,A -85,B 0,C 180,E1 -4571.221,E2 -4571.221} C_VEL
LIN {X 0,Y 523.936,Z 91.529,A -85,B 0,C 180,E1 -4573.639,E2 -4573.639} C_VEL
LIN {X 0,Y 523.94,Z 91.533,A -85,B 0,C 180,E1 -4576.029,E2 -4576.029} C_VEL
LIN {X 0,Y 524.012,Z 91.526,A -85,B 0,C 180,E1 -4578.395,E2 -4578.395} C_VEL
LIN {X 0,Y 524.004,Z 91.521,A -85,B 0,C 180,E1 -4581.517,E2 -4581.517} C_VEL
LIN {X 0,Y 524.082,Z 91.513,A -85,B 0,C 180,E1 -4584.614,E2 -4584.614} C_VEL
LIN {X 0,Y 524.112,Z 91.51,A -85,B 0,C 180,E1 -4587.695,E2 -4587.695} C_VEL
LIN {X 0,Y 524.124,Z 91.506,A -85,B 0,C 180,E1 -4590.769,E2 -4590.769} C_VEL
LIN {X 0,Y 524.071,Z 91.512,A -85,B 0,C 180,E1 -4593.075,E2 -4593.075} C_VEL
LIN {X 0,Y 524.047,Z 91.521,A -85,B 0,C 180,E1 -4596.16,E2 -4596.16} C_VEL
LIN {X 0,Y 523.999,Z 91.522,A -85,B 0,C 180,E1 -4599.262,E2 -4599.262} C_VEL
LIN {X 0,Y 524.005,Z 91.527,A -85,B 0,C 180,E1 -4601.74,E2 -4601.74} C_VEL
LIN {X 0,Y 523.995,Z 91.522,A -85,B 0,C 180,E1 -4605.053,E2 -4605.053} C_VEL
LIN {X 0,Y 523.966,Z 91.531,A -85,B 0,C 180,E1 -4607.969,E2 -4607.969} C_VEL
LIN {X 0,Y 523.974,Z 91.525,A -85,B 0,C 180,E1 -4610.41,E2 -4610.41} C_VEL
LIN {X 0,Y 523.913,Z 91.532,A -85,B 0,C 180,E1 -4612.894,E2 -4612.894} C_VEL
LIN {X 0,Y 523.987,Z 91.525,A -85,B 0,C 180,E1 -4616.02,E2 -4616.02} C_VEL
LIN {X 0,Y 523.941,Z 91.529,A -85,B 0,C 180,E1 -4618.875,E2 -4618.875} C_VEL
LIN {X 0,Y 523.926,Z 91.539,A -85,B 0,C 180,E1 -4621.544,E2 -4621.544} C_VEL
LIN {X 0,Y 523.935,Z 91.529,A -85,B 0,C 180,E1 -4624.291,E2 -4624.291} C_VEL
LIN {X 0,Y 523.909,Z 91.537,A -85,B 0,C 180,E1 -4627.133,E2 -4627.133} C_VEL
LIN {X 0,Y 523.94,Z 91.528,A -85,B 0,C 180,E1 -4630.13,E2 -4630.13} C_VEL
LIN {X 0,Y 523.938,Z 91.528,A -85,B 0,C 180,E1 -4632.459,E2 -4632.459} C_VEL
LIN {X 0,Y 523.953,Z 91.535,A -85,B 0,C 180,E1 -4635.31,E2 -4635.31} C_VEL
LIN {X 0,Y 523.958,Z 91.528,A -85,B 0,C 180,E1 -4638.69,E2 -4638.69} C_VEL
LIN {X 0,Y 523.921,Z 91.538,A -85,B 0,C 180,E1 -4641.081,E2 -4641.081} C_VEL
LIN {X 0,Y 523.909,Z 91.534,A -85,B 0,C 180,E1 -4643.826,E2 -4643.826} C_VEL
LIN {X 0,Y 523.945,Z 91.531,A -85,B 0,C 180,E1 -4646.636,E2 -4646.636} C_VEL
LIN {X 0,Y 523.959,Z 91.532,A -85,B 0,C 180,E1 -4649.356,E2 -4649.356} C_VEL
LIN {X 0,Y 523.981,Z 91.528,A -85,B 0,C 180,E1 -4652.282,E2 -4652.282} C_VEL
LIN {X 0,Y 523.987,Z 91.528,A -85,B 0,C 180,E1 -4654.081,E2 -4654.081} C_VEL
LIN {X 0,Y 525.041,Z 94.485,A -85,B 0,C 180,E1 -4654.193,E2 -4654.193} C_VEL
LIN {X 0,Y 530.655,Z 106.292,A -85,B 0,C 180,E1 -4654.677,E2 -4654.677} C_VEL
LIN {X 0,Y 529.838,Z 190.17,A -85,B 0,C 180,E1 -4655.946,E2 -4655.946} C_VEL
LIN {X 0,Y 528.95,Z 288.812,A -85,B 0,C 180,E1 -4657.414,E2 -4657.414} C_VEL
LIN {X 0,Y 528.624,Z 305.345,A -85,B 0,C 180,E1 -4657.811,E2 -4657.811} C_VEL
LIN {X 0,Y 528.235,Z 321.261,A -85,B 0,C 180,E1 -4658.346,E2 -4658.346} C_VEL
LIN {X 0,Y 527.794,Z 336.97,A -85,B 0,C 180,E1 -4659.031,E2 -4659.031} C_VEL
LIN {X 0,Y 527.273,Z 351.685,A -85,B 0,C 180,E1 -4659.825,E2 -4659.825} C_VEL
LIN {X 0,Y 526.666,Z 366.74,A -85,B 0,C 180,E1 -4660.816,E2 -4660.816} C_VEL
LIN {X 0,Y 526.115,Z 379.8,A -85,B 0,C 180,E1 -4661.849,E2 -4661.849} C_VEL
LIN {X 0,Y 525.594,Z 391.135,A -85,B 0,C 180,E1 -4662.892,E2 -4662.892} C_VEL
LIN {X 0,Y 525.154,Z 402.264,A -85,B 0,C 180,E1 -4664.077,E2 -4664.077} C_VEL
LIN {X 0,Y 524.67,Z 413.343,A -85,B 0,C 180,E1 -4665.454,E2 -4665.454} C_VEL
LIN {X 0,Y 524.272,Z 424.005,A -85,B 0,C 180,E1 -4667.024,E2 -4667.024} C_VEL
LIN {X 0,Y 523.939,Z 432.857,A -85,B 0,C 180,E1 -4668.589,E2 -4668.589} C_VEL
LIN {X 0,Y 523.696,Z 439.414,A -85,B 0,C 180,E1 -4669.953,E2 -4669.953} C_VEL
LIN {X 0,Y 523.557,Z 445.666,A -85,B 0,C 180,E1 -4671.509,E2 -4671.509} C_VEL
LIN {X 0,Y 523.476,Z 451.819,A -85,B 0,C 180,E1 -4673.465,E2 -4673.465} C_VEL
LIN {X 0,Y 523.399,Z 454.652,A -85,B 0,C 180,E1 -4674.607,E2 -4674.607} C_VEL
LIN {X 0,Y 523.402,Z 457.513,A -85,B 0,C 180,E1 -4676.15,E2 -4676.15} C_VEL
LIN {X 0,Y 523.328,Z 459.423,A -85,B 0,C 180,E1 -4677.691,E2 -4677.691} C_VEL
LIN {X 0,Y 523.264,Z 460.381,A -85,B 0,C 180,E1 -4679.23,E2 -4679.23} C_VEL
LIN {X 0,Y 523.266,Z 460.421,A -85,B 0,C 180,E1 -4680.769,E2 -4680.769} C_VEL
LIN {X 0,Y 523.329,Z 459.53,A -85,B 0,C 180,E1 -4682.309,E2 -4682.309} C_VEL
LIN {X 0,Y 523.416,Z 457.689,A -85,B 0,C 180,E1 -4683.849,E2 -4683.849} C_VEL
LIN {X 0,Y 523.402,Z 454.917,A -85,B 0,C 180,E1 -4685.393,E2 -4685.393} C_VEL
LIN {X 0,Y 523.547,Z 449.918,A -85,B 0,C 180,E1 -4687.327,E2 -4687.327} C_VEL
LIN {X 0,Y 523.59,Z 444.706,A -85,B 0,C 180,E1 -4688.88,E2 -4688.88} C_VEL
LIN {X 0,Y 523.825,Z 438.266,A -85,B 0,C 180,E1 -4690.435,E2 -4690.435} C_VEL
LIN {X 0,Y 524.124,Z 429.387,A -85,B 0,C 180,E1 -4692.192,E2 -4692.192} C_VEL
LIN {X 0,Y 524.466,Z 419.759,A -85,B 0,C 180,E1 -4693.76,E2 -4693.76} C_VEL
LIN {X 0,Y 524.824,Z 410.639,A -85,B 0,C 180,E1 -4695.028,E2 -4695.028} C_VEL
LIN {X 0,Y 525.281,Z 399.778,A -85,B 0,C 180,E1 -4696.318,E2 -4696.318} C_VEL
LIN {X 0,Y 525.812,Z 387.08,A -85,B 0,C 180,E1 -4697.602,E2 -4697.602} C_VEL
LIN {X 0,Y 526.337,Z 374.387,A -85,B 0,C 180,E1 -4698.691,E2 -4698.691} C_VEL
LIN {X 0,Y 526.878,Z 360.686,A -85,B 0,C 180,E1 -4699.682,E2 -4699.682} C_VEL
LIN {X 0,Y 527.372,Z 345.694,A -85,B 0,C 180,E1 -4700.578,E2 -4700.578} C_VEL
LIN {X 0,Y 527.843,Z 330.053,A -85,B 0,C 180,E1 -4701.334,E2 -4701.334} C_VEL
LIN {X 0,Y 528.237,Z 313.76,A -85,B 0,C 180,E1 -4701.949,E2 -4701.949} C_VEL
LIN {X 0,Y 528.515,Z 297.683,A -85,B 0,C 180,E1 -4702.399,E2 -4702.399} C_VEL
LIN {X 0,Y 528.697,Z 281.949,A -85,B 0,C 180,E1 -4702.7,E2 -4702.7} C_VEL
LIN {X 0,Y 529.932,Z 165.704,A -85,B 0,C 180,E1 -4704.457,E2 -4704.457} C_VEL
LIN {X 0,Y 530.653,Z 106.266,A -85,B 0,C 180,E1 -4705.43,E2 -4705.43} C_VEL
LIN {X 0,Y 524.851,Z 94.301,A -85,B 0,C 180,E1 -4705.977,E2 -4705.977} C_VEL
LIN {X 0,Y 523.879,Z 91.543,A -85,B 0,C 180,E1 -4706.097,E2 -4706.097} C_VEL
LIN {X 0,Y 523.899,Z 91.542,A -85,B 0,C 180,E1 -4708.877,E2 -4708.877} C_VEL
LIN {X 0,Y 523.911,Z 91.537,A -85,B 0,C 180,E1 -4711.545,E2 -4711.545} C_VEL
LIN {X 0,Y 523.921,Z 91.538,A -85,B 0,C 180,E1 -4714.291,E2 -4714.291} C_VEL
LIN {X 0,Y 523.906,Z 91.537,A -85,B 0,C 180,E1 -4717.132,E2 -4717.132} C_VEL
LIN {X 0,Y 523.94,Z 91.536,A -85,B 0,C 180,E1 -4720.129,E2 -4720.129} C_VEL
LIN {X 0,Y 523.936,Z 91.537,A -85,B 0,C 180,E1 -4722.458,E2 -4722.458} C_VEL
LIN {X 0,Y 523.947,Z 91.531,A -85,B 0,C 180,E1 -4725.309,E2 -4725.309} C_VEL
LIN {X 0,Y 523.957,Z 91.53,A -85,B 0,C 180,E1 -4728.689,E2 -4728.689} C_VEL
LIN {X 0,Y 523.918,Z 91.535,A -85,B 0,C 180,E1 -4731.08,E2 -4731.08} C_VEL
LIN {X 0,Y 523.902,Z 91.543,A -85,B 0,C 180,E1 -4733.825,E2 -4733.825} C_VEL
LIN {X 0,Y 523.943,Z 91.538,A -85,B 0,C 180,E1 -4736.635,E2 -4736.635} C_VEL
LIN {X 0,Y 523.943,Z 91.545,A -85,B 0,C 180,E1 -4738.372,E2 -4738.372} C_VEL
LIN {X 0,Y 528.892,Z 107.894,A -85,B 0,C 180,E1 -4740.201,E2 -4740.201} C_VEL
LIN {X 0,Y 528.916,Z 114.443,A -85,B 0,C 180,E1 -4740.791,E2 -4740.791} C_VEL
LIN {X 0,Y 527.928,Z 145.183,A -85,B 0,C 180,E1 -4743.427,E2 -4743.427} C_VEL
LIN {X 0,Y 527.811,Z 152.903,A -85,B 0,C 180,E1 -4744.062,E2 -4744.062} C_VEL
LIN {X 0,Y 530.504,Z 172.593,A -85,B 0,C 180,E1 -4744.538,E2 -4744.538} C_VEL
LIN {X 0,Y 529.039,Z 292.327,A -85,B 0,C 180,E1 -4746.384,E2 -4746.384} C_VEL
LIN {X 0,Y 528.455,Z 363.788,A -85,B 0,C 180,E1 -4747.443,E2 -4747.443} C_VEL
LIN {X 0,Y 528.086,Z 381.379,A -85,B 0,C 180,E1 -4747.864,E2 -4747.864} C_VEL
LIN {X 0,Y 527.631,Z 398.383,A -85,B 0,C 180,E1 -4748.44,E2 -4748.44} C_VEL
LIN {X 0,Y 527.171,Z 414.042,A -85,B 0,C 180,E1 -4749.128,E2 -4749.128} C_VEL
